// TwinCAT 3 PLC project CORE
// Title: ZigaLibs.Core
// Company: Ziga Javornik
// Author: Ziga Javornik
// ProjectVersion: 0.0.3.7
// Description: A collection of core objects for work with further libraries implementations.
// ProgramVersion: 3.1.4026.26
// libraries:
//   Tc2_EtherCAT, * (Beckhoff Automation GmbH)
//   Tc2_IoFunctions, * (Beckhoff Automation GmbH)
//   Tc2_Standard, * (Beckhoff Automation GmbH)
//   Tc2_System, * (Beckhoff Automation GmbH)
//   Tc2_Utilities, * (Beckhoff Automation GmbH)
//   Tc3_Module, * (Beckhoff Automation GmbH)
//   TcError, * (Roald87)
//   TcUnit, * (www.tcunit.org)
//   Base Interfaces,newest,System
// project tree:
//   SOURCE/Array/ ArrayHelper.TcPOU
//   SOURCE/Array/DUTs/ ST_ArrayProperties.TcDUT, T_ArrayIndexer.TcDUT
//   SOURCE/Beckhoff/Ads/ AdsHelper.TcPOU, FB_HasAmsAddressFromProcessImage.TcPOU, I_HasAmsAddress.TcIO
//   SOURCE/Beckhoff/EtherCAT/CoE/DUTs/ ST_CoeEntry.TcDUT, ST_CoeEntry_DINT.TcDUT, ST_CoeEntry_SINT.TcDUT, ST_CoeEntry_String128.TcDUT, ST_CoeEntry_UDINT.TcDUT, ST_CoeEntry_INT.TcDUT, ST_CoeEntry_REAL.TcDUT, ST_CoeEntry_String255.TcDUT, ST_CoeEntry_String30.TcDUT, ST_CoeEntry_UINT.TcDUT, ST_CoeEntry_USINT.TcDUT, T_CoEIndex.TcDUT, T_CoESubIndex.TcDUT
//   SOURCE/Beckhoff/EtherCAT/CoE/ FB_CoeReadWrite.TcPOU, I_ReadsCoE.TcIO
//   SOURCE/Beckhoff/EtherCAT/Diagnosis/DUTs/Device state/ E_EcDeviceState.TcDUT, E_EcDeviceStateExtras.TcDUT, E_EcLinkState.TcDUT, ST_EcDeviceState.TcDUT, ST_EcSlaveState.TcDUT
//   SOURCE/Beckhoff/EtherCAT/Diagnosis/DUTs/ E_EthercatDiagnosisState.TcDUT, E_EthercatDiagnosisStatus.TcDUT, ST_EthercatSlaveInfo.TcDUT
//   SOURCE/Beckhoff/EtherCAT/Diagnosis/ FB_EthercatDiagnosis.TcPOU (excluded from build), I_EthercatDiagnosis.TcIO
//   SOURCE/Beckhoff/EtherCAT/ EthercatHelper.TcPOU, FB_ReadBoxName.TcPOU
//   SOURCE/Errors/DUTs/ ST_AdsError.TcDUT, ST_Error.TcDUT, ST_GenericError.TcDUT
//   SOURCE/Errors/ FB_ErrorSource.TcPOU, I_HasError.TcIO, I_ErrorSource.TcIO, I_HasAdsError.TcIO, I_HasGenericError.TcIO
//   SOURCE/General/ FB_BooleanObserver.TcPOU, FB_HasInstanceNameAndPath.TcPOU, FB_HasTaskInfo.TcPOU, FB_Watchdog.TcPOU, InstanceNameHelper.TcPOU, ST_Value.TcDUT (not stored)
//   SOURCE/General/Memory/ FB_Malloc.TcPOU, MemoryHelper.TcPOU, ST_AllocatedMemoryProperties.TcDUT, E_MemCmpResults.TcDUT
//   SOURCE/General/Variable information/ T_VarInfo.TcDUT, F_DoesVarTypeEqual.TcPOU, F_GetVarInfo.TcPOU, ST_VarInfo.TcDUT, T_VarSize.TcDUT
//   SOURCE/General/Variable extensions/ BoolEx.TcPOU
//   SOURCE/String/StringBuilder/Extensions/AddAny/ E_AddAnyBitOptions.TcDUT, I_StringBuilderEx_Any.TcIO
//   SOURCE/String/StringBuilder/ FB_StringBuilder.TcPOU, I_StringBuilder.TcIO
//   SOURCE/String/ StringConstants.TcPOU, StringHelper.TcPOU, T_Char.TcDUT
//   SOURCE/Time/DUTs/ E_TimeFormat.TcDUT (not stored), ST_CurrentSystemTimeInfo.TcDUT
//   SOURCE/Time/ FB_DateTimeToStringConverter.TcPOU, FB_LocalSystemTimeProvider.TcPOU, I_DateTimeToStringConverter.TcIO, I_LocalSystemTimeProvider.TcIO
//   / TestsTask.TcTTO
//   TESTS/ PRG_TESTS.TcPOU
//   TESTS/Test suites/ FB_AdsHelper_Tests.TcPOU, FB_ArrayHelper_Tests.TcPOU, FB_CoeReadWrite_Tests.TcPOU, FB_DateTimeToStringConverter_Tests.TcPOU, FB_ErrorSource_ExtensionForTests.TcPOU, FB_ErrorSource_Tests.TcPOU, FB_EthercatDiagnosis_Tests.TcPOU (excluded from build), FB_EthercatHelper_Tests.TcPOU, FB_HasInstanceName_ExtensionForTests.TcPOU, FB_HasInstanceName_Tests.TcPOU, FB_HasTaskInfo_ExtensionsForTests.TcPOU, FB_HasTaskInfo_Tests.TcPOU, FB_Malloc_Tests.TcPOU, FB_StringBuilderEx_Any_Tests.TcPOU, FB_StringBuilder_Tests.TcPOU, FB_BoolEx_Tests.TcPOU, FB_StringHelper_Tests.TcPOU
//   TESTS/Test suites/Time/ FB_LocalSystemTime_Tests.TcPOU
// (motion and I/O tree: see PLC project logging)
// real-time tasks:
//   TASK TestsTask: cycle T#10ms, priority 20, ADS port 350
//   TASK PlcTask: cycle T#10ms, priority 21, ADS port 351

CONFIGURATION CORE
    RESOURCE PLC ON TwinCAT3
        TASK TestsTask(INTERVAL := T#10ms, PRIORITY := 20);
        PROGRAM PRG_TESTS WITH TestsTask : PRG_TESTS;
    END_RESOURCE
END_CONFIGURATION

// ---- SOURCE/Array/DUTs/ST_ArrayProperties.TcDUT
TYPE ST_ArrayProperties :
STRUCT
	Count		: DINT;
	StartIndex	: T_ArrayIndexer;
	EndIndex	: T_ArrayIndexer;
END_STRUCT
END_TYPE

// ---- SOURCE/Array/DUTs/T_ArrayIndexer.TcDUT
// Should be used when accessing array index.
TYPE T_ArrayIndexer : DINT; END_TYPE

// ---- SOURCE/Beckhoff/EtherCAT/CoE/DUTs/ST_CoeEntry.TcDUT
{attribute 'qualified_only'}
// CoE entry in the dictionary, includes index and the subindex
TYPE ST_CoeEntry :
STRUCT
	Index		: T_CoEIndex;
	Subindex	: T_CoESubIndex;
END_STRUCT
END_TYPE

// ---- SOURCE/Beckhoff/EtherCAT/CoE/DUTs/ST_CoeEntry_DINT.TcDUT
TYPE ST_CoeEntry_DINT EXTENDS ST_CoeEntry :
STRUCT
	Value	: DINT;
END_STRUCT
END_TYPE

// ---- SOURCE/Beckhoff/EtherCAT/CoE/DUTs/ST_CoeEntry_SINT.TcDUT
TYPE ST_CoeEntry_SINT EXTENDS ST_CoeEntry :
STRUCT
	Value	: SINT;
END_STRUCT
END_TYPE

// ---- SOURCE/Beckhoff/EtherCAT/CoE/DUTs/ST_CoeEntry_String128.TcDUT
TYPE ST_CoeEntry_String128 EXTENDS ST_CoeEntry :
STRUCT
	Value	: STRING(128);
END_STRUCT
END_TYPE

// ---- SOURCE/Beckhoff/EtherCAT/CoE/DUTs/ST_CoeEntry_UDINT.TcDUT
TYPE ST_CoeEntry_UDINT EXTENDS ST_CoeEntry :
STRUCT
	Value	: UDINT;
END_STRUCT
END_TYPE

// ---- SOURCE/Beckhoff/EtherCAT/CoE/DUTs/ST_CoeEntry_INT.TcDUT
TYPE ST_CoeEntry_INT EXTENDS ST_CoeEntry :
STRUCT
	Value	: INT;
END_STRUCT
END_TYPE

// ---- SOURCE/Beckhoff/EtherCAT/CoE/DUTs/ST_CoeEntry_REAL.TcDUT
TYPE ST_CoeEntry_REAL EXTENDS ST_CoeEntry :
STRUCT
	Value	: REAL;
END_STRUCT
END_TYPE

// ---- SOURCE/Beckhoff/EtherCAT/CoE/DUTs/ST_CoeEntry_String255.TcDUT
TYPE ST_CoeEntry_String255 EXTENDS ST_CoeEntry :
STRUCT
	Value	: Tc2_System.T_MaxString;
END_STRUCT
END_TYPE

// ---- SOURCE/Beckhoff/EtherCAT/CoE/DUTs/ST_CoeEntry_String30.TcDUT
TYPE ST_CoeEntry_String30 EXTENDS ST_CoeEntry :
STRUCT
	Value	: STRING(30);
END_STRUCT
END_TYPE

// ---- SOURCE/Beckhoff/EtherCAT/CoE/DUTs/ST_CoeEntry_UINT.TcDUT
TYPE ST_CoeEntry_UINT EXTENDS ST_CoeEntry :
STRUCT
	Value	: UINT;
END_STRUCT
END_TYPE

// ---- SOURCE/Beckhoff/EtherCAT/CoE/DUTs/ST_CoeEntry_USINT.TcDUT
TYPE ST_CoeEntry_USINT EXTENDS ST_CoeEntry :
STRUCT
	Value	: USINT;
END_STRUCT
END_TYPE

// ---- SOURCE/Beckhoff/EtherCAT/CoE/DUTs/T_CoEIndex.TcDUT
TYPE T_CoEIndex : WORD; END_TYPE

// ---- SOURCE/Beckhoff/EtherCAT/CoE/DUTs/T_CoESubIndex.TcDUT
TYPE T_CoESubIndex : BYTE; END_TYPE

// ---- SOURCE/Beckhoff/EtherCAT/Diagnosis/DUTs/Device state/E_EcDeviceState.TcDUT
{attribute 'qualified_only'}
TYPE E_EcDeviceState :
(
	INIT		:= Tc2_EtherCAT.EC_DEVICE_STATE_INIT,
	PREOP		:= Tc2_EtherCAT.EC_DEVICE_STATE_PREOP,
	BOOTSTRAP	:= Tc2_EtherCAT.EC_DEVICE_STATE_BOOTSTRAP,
	SAFEOP		:= Tc2_EtherCAT.EC_DEVICE_STATE_SAFEOP,
	OP			:= Tc2_EtherCAT.EC_DEVICE_STATE_OP
)BYTE;
END_TYPE

// ---- SOURCE/Beckhoff/EtherCAT/Diagnosis/DUTs/Device state/E_EcDeviceStateExtras.TcDUT
{attribute 'qualified_only'}
TYPE E_EcDeviceStateExtras :
(
	NOTHING				:= 16#00,
	STATE_MACHINE_ERROR := Tc2_EtherCAT.EC_DEVICE_STATE_ERROR,
	INVALID_VPRS		:= Tc2_EtherCAT.EC_DEVICE_STATE_INVALID_VPRS,
	INIIT_CMD_ERROR		:= Tc2_EtherCAT.EC_DEVICE_STATE_INITCMD_ERROR,
	DISABLED			:= Tc2_EtherCAT.EC_DEVICE_STATE_DISABLED
)BYTE;
END_TYPE

// ---- SOURCE/Beckhoff/EtherCAT/Diagnosis/DUTs/Device state/E_EcLinkState.TcDUT
TYPE E_EcLinkState :
(
	OK					:= Tc2_EtherCAT.EC_LINK_STATE_OK,
	NOT_PRESENT			:= Tc2_EtherCAT.EC_LINK_STATE_NOT_PRESENT,
	LINK_WITHOUT_COMM	:= Tc2_EtherCAT.EC_LINK_STATE_LINK_WITHOUT_COMM,
	MISSING_LINK		:= Tc2_EtherCAT.EC_LINK_STATE_MISSING_LINK,
	ADDITIONAL_LINK		:= Tc2_EtherCAT.EC_LINK_STATE_ADDITIONAL_LINK,
	PORT_A				:= Tc2_EtherCAT.EC_LINK_STATE_PORT_A,
	PORT_B				:= Tc2_EtherCAT.EC_LINK_STATE_PORT_B,
	PORT_C				:= Tc2_EtherCAT.EC_LINK_STATE_PORT_C,
	PORT_D				:= Tc2_EtherCAT.EC_LINK_STATE_PORT_D
)BYTE;
END_TYPE

// ---- SOURCE/Beckhoff/EtherCAT/Diagnosis/DUTs/Device state/ST_EcDeviceState.TcDUT
TYPE ST_EcDeviceState :
STRUCT
	State		: E_EcDeviceState;	// Device state
	StateExtras	: E_EcDeviceStateExtras;	// Extra information
END_STRUCT
END_TYPE

// ---- SOURCE/Beckhoff/EtherCAT/Diagnosis/DUTs/Device state/ST_EcSlaveState.TcDUT
TYPE ST_EcSlaveState :
STRUCT
	Device	: ST_EcDeviceState;	// Device state
	Link	: E_EcLinkState;	// Link state
END_STRUCT
END_TYPE

// ---- SOURCE/Beckhoff/EtherCAT/Diagnosis/DUTs/E_EthercatDiagnosisState.TcDUT
{attribute 'qualified_only'}
{attribute 'strict'}
TYPE E_EthercatDiagnosisState :
(
	READY,
	GET_SLAVE_STATES,
	GET_FAULTY_SLAVE_ADDRESSES,
	FINISHED,
	ERROR
);
END_TYPE

// ---- SOURCE/Beckhoff/EtherCAT/Diagnosis/DUTs/E_EthercatDiagnosisStatus.TcDUT
TYPE E_EthercatDiagnosisStatus :
(
	NO_ERROR,				// No error, all slaves are present
	MISSING_ALLOWED_SLAVES,	// Missing slaves, but they are allowed (for example, hot connect)
	ERROR					// Missing slaves that are not allowed to be missing
);
END_TYPE

// ---- SOURCE/Beckhoff/EtherCAT/Diagnosis/DUTs/ST_EthercatSlaveInfo.TcDUT
TYPE ST_EthercatSlaveInfo :
STRUCT
	Name		: Tc2_System.T_MaxString;	// Slave name
	IsIgnored	: BOOL;	// True if slave is ignored with the scan
	State		: ST_EcSlaveState;
END_STRUCT
END_TYPE

// ---- SOURCE/Errors/DUTs/ST_AdsError.TcDUT
TYPE ST_AdsError EXTENDS ST_Error:
STRUCT
	Code	: TcError.AdsErrorCodes;
	Message	: Tc2_System.T_MaxString;
END_STRUCT
END_TYPE

// ---- SOURCE/Errors/DUTs/ST_Error.TcDUT
TYPE ST_Error :
STRUCT
	Source	: Tc2_System.T_MaxString;
END_STRUCT
END_TYPE

// ---- SOURCE/Errors/DUTs/ST_GenericError.TcDUT
TYPE ST_GenericError EXTENDS ST_Error :
STRUCT
	Code	: DINT;
	Message	: Tc2_System.T_MaxString;
END_STRUCT
END_TYPE

// ---- SOURCE/General/Memory/ST_AllocatedMemoryProperties.TcDUT
// Properties for working with dynamic memory allocation.
TYPE ST_AllocatedMemoryProperties :
STRUCT
	Size				: DINT;		// Size of the allocated memory
	StartAddress		: PVOID;	// Pointer to the address of the array memory space
	BaseTypeSize		: DINT;		// Size of the base type provided, when allocated
	NumberOfElements	: DINT;	// Number of elements provided, when allocated.
END_STRUCT
END_TYPE

// ---- SOURCE/General/Variable information/T_VarInfo.TcDUT
TYPE T_VarInfo : __SYSTEM.VAR_INFO; END_TYPE

// ---- SOURCE/General/Memory/E_MemCmpResults.TcDUT
{attribute 'qualified_only'}
TYPE E_MemCmpResults :
(
	pBUFF1_LESS_THAN_pBUFF2	:= -1,
	IDENTICAL	:= 0,
	PbUFF1_GREATER_THAN_pBUFF2	:= 1,
	ERROR	:= 255
)DINT;
END_TYPE

// ---- SOURCE/General/Variable information/ST_VarInfo.TcDUT
TYPE ST_VarInfo :
STRUCT
	DataType	: __SYSTEM.TYPE_CLASS;
	Address		: POINTER TO BYTE;
	Size		: T_VarSize;
END_STRUCT
END_TYPE

// ---- SOURCE/General/Variable information/T_VarSize.TcDUT
// Variable size alias type. To be used when working with SIZEOF operator.
TYPE T_VarSize : UXINT; END_TYPE

// ---- SOURCE/String/StringBuilder/Extensions/AddAny/E_AddAnyBitOptions.TcDUT
{attribute 'qualified_only'}
{attribute 'strict'}
// Provides various options of how ANY_BIT data type can be converted.
TYPE E_AddAnyBitOptions :
(
	BINARY,			// Will be converted to a binary string (base 2)
	DECIMAL,		// Will be converted to a decial string (base 10)
	HEXADECIMAL,	// Will be converted to hexadecimal string (base 16)
	OCTAL			// Will be converted to octal string (base 8)
);
END_TYPE

// ---- SOURCE/String/T_Char.TcDUT
TYPE T_Char : STrING(1); END_TYPE

// ---- SOURCE/Time/DUTs/ST_CurrentSystemTimeInfo.TcDUT
TYPE ST_CurrentSystemTimeInfo :
STRUCT
	IsValid	: BOOL;
	Value	: Tc2_Utilities.TIMESTRUCT;
END_STRUCT
END_TYPE

// ---- SOURCE/Beckhoff/Ads/I_HasAmsAddress.TcIO
// Interface to implement when requiring AMS address
INTERFACE I_HasAmsAddress

// Gets or sets the Ams address structure
PROPERTY AmsAddress : REFERENCE TO Tc2_System.ST_AmsAddr
GET
END_GET
SET
END_SET
END_PROPERTY

END_INTERFACE

// ---- SOURCE/Beckhoff/EtherCAT/CoE/I_ReadsCoE.TcIO
INTERFACE I_ReadsCoE

// Reads CoE items and updates them. Returns TRUE when done,
// Needs to be called until the method finishes, indicating via the return value. 
METHOD PUBLIC ReadCoE : BOOL
END_METHOD

END_INTERFACE

// ---- SOURCE/Beckhoff/EtherCAT/Diagnosis/I_EthercatDiagnosis.TcIO
INTERFACE I_EthercatDiagnosis

// Returns TRUE if an error occurred while performing the scan
PROPERTY Error : BOOL
GET
END_GET
END_PROPERTY

// Gets an array of slaves that have been added to ignore list
PROPERTY IgnoredSlaves : REFERENCE TO ARRAY[0..255] OF Tc2_System.T_MaxString
GET
END_GET
END_PROPERTY

// Adds the provided slave to a collection of slaves that will not trigger an error
// Example is slaves that are used on hot connect groups, and when connected should not cause an error. 
METHOD IgnoreSlave
VAR_INPUT
	Name	: Tc2_System.T_MaxString;	// Slave to be ignored if not found or an error is reported back
END_VAR
END_METHOD

// Returns an array of misisng slave names
PROPERTY MissingSlaves : REFERENCE TO ARRAY[0..255] OF ST_EthercatSlaveInfo
GET
END_GET
END_PROPERTY

// Reset the internal state machine of diagnosis and clearing any errors, if active.
METHOD Reset
END_METHOD

// Performs a scan on the EtherCAT master, returns TRUE when done.
METHOD Scan	: BOOL
VAR_INPUT
	EcMasterNetId	: AMSNETID;
END_VAR
END_METHOD

// Gets the status based on last executed scan.
PROPERTY Status : E_EthercatDiagnosisStatus
GET
END_GET
END_PROPERTY

END_INTERFACE

// ---- SOURCE/Errors/I_HasError.TcIO
INTERFACE I_HasError

{attribute 'monitoring':='call'}
// Returns TRUE if an error has occurred
PROPERTY Error : BOOL
GET
END_GET
END_PROPERTY

END_INTERFACE

// ---- SOURCE/Errors/I_ErrorSource.TcIO
INTERFACE I_ErrorSource EXTENDS I_HasAdsError, I_HasGenericError, I_HasError

END_INTERFACE

// ---- SOURCE/Errors/I_HasAdsError.TcIO
INTERFACE I_HasAdsError

{attribute 'monitoring':='call'}
// Gets or sets the Ads error - note that code to message conversion is done automatically.
PROPERTY AdsError : REFERENCE TO ST_AdsError
GET
END_GET
END_PROPERTY

END_INTERFACE

// ---- SOURCE/Errors/I_HasGenericError.TcIO
INTERFACE I_HasGenericError

{attribute 'monitoring':='call'}
// Gets the Generic error
PROPERTY GenericError : REFERENCE TO ST_GenericError
GET
END_GET
END_PROPERTY

END_INTERFACE

// ---- SOURCE/String/StringBuilder/Extensions/AddAny/I_StringBuilderEx_Any.TcIO
INTERFACE I_StringBuilderEx_Any

(* Adds the variable of any data type to the sequence. Conversion is done automatically from within.
Some extra info: 
	- BOOL and BIT will have the string converted to 'TRUE' and 'FALSE' respectively.
	- floating point variables will have their values precision based on constructor realFormatPrecision and will be rounded based on the roundRealValues
*)
METHOD AddAny : REFERENCE TO FB_StringBuilder
VAR_INPUT
	anyVar	: ANY;
END_VAR
END_METHOD

// Adds a variable of type ANY_BIT to the string generating sequence, based on the provided parameters.
// This includes: BYTE, WORD, DWORD, LWORD, 
METHOD AddAnyBit : REFERENCE TO FB_StringBuilder
VAR_INPUT
	anyBit					: ANY_BIT;				// Value to be converterd
	option					: E_AddAnyBitOptions;	// Select how the value is converter
	lowerCase				: BOOL;					// If hexadecimal option is selected, the result string can be converted to either lower or upper case
	displayedDigitsCount	: INT;					// This determines how many digits are to be displayed. If actual digits count is lower, the string is filled with zeros from the left side. If left at 0, the result string will be an empty string!
	addNotation				: BOOL;					// If this is set to TRUE, a notation will be prepended: (DEC)10, (BIN)10, (HEX)10, (OCT)10
END_VAR
END_METHOD

// Adds any REAL or LREAL value to the generating string sequence.
// Please note that REAL values will ALWAYS be automatically rounded on 3rd decimal digit.
// Anything after it will be whatever TwinCAT representation decides to do.
METHOD AddAnyReal : REFERENCE TO FB_StringBuilder
VAR_INPUT
	anyReal		: ANY_REAL;	// Value to be converter
	precision	: INT;		// Precision
	round		: BOOL;		// Rounding of the last displayed digit
END_VAR
END_METHOD

END_INTERFACE

// ---- SOURCE/String/StringBuilder/I_StringBuilder.TcIO
INTERFACE I_StringBuilder

// Adds a string to the build sequence.
METHOD AddString : REFERENCE TO FB_StringBuilder
VAR_INPUT
	str	: Tc2_System.T_MaxString;	// String to be added.
END_VAR
END_METHOD

// Adds a string to the build sequence and wraps the str in double quotation marks "str"
METHOD AddWithDblQuotationMarks : REFERENCE TO FB_StringBuilder
VAR_INPUT
	str : Tc2_System.T_MaxString;
END_VAR
END_METHOD

// Adds a string to the build sequence and wraps the str in quotation marks 'str'
METHOD AddWithQuotationMark : REFERENCE TO FB_StringBuilder
VAR_INPUT
	str	: Tc2_System.T_MaxString;
END_VAR
END_METHOD

// Finishes string generation and returns the generated string
METHOD Create : Tc2_System.T_MaxString
END_METHOD

(* Reset the string build sequence, clear any string built so far.*)
METHOD Reset : REFERENCE TO FB_StringBuilder
VAR_INPUT
END_VAR
END_METHOD

END_INTERFACE

// ---- SOURCE/Time/I_DateTimeToStringConverter.TcIO
INTERFACE I_DateTimeToStringConverter

(* Converts TIMESTRUCT to STRING.*)
METHOD DateTime : STRING
VAR_INPUT
	timeFormat			: E_TimeFormat;	// Time format to apply to the timestruct conversion
	timeOfDaySeperator	: STRING(1);	// Specifies how time of day is split
	dateSeperator		: STRING(1);	// Specifies how date is split
	fillWithZeros		: BOOL;	// If set to true: month, day hour, minute and second will have 0 added when only a single digit is present
	IncludeMilliseconds	: BOOL; // If set to true, milliseconds will also be displayed in the result, else they are ignored
END_VAR
END_METHOD

(* Converts TIMESTRUCT.wDay to STRING.*)
METHOD Day : STRING
VAR_INPUT
	fillWithZeros	: BOOL;	// If set to true, result will have 0 added when only a single digit is present
END_VAR
END_METHOD

(* Converts TIMESTRUCT.wHour to STRING.*)
METHOD Hour : STRING
VAR_INPUT
	fillWithZeros	: BOOL;	// If set to true, result will have 0 added when only a single digit is present
END_VAR
END_METHOD

(* Converts TIMESTRUCT.wMillisecond to STRING.*)
METHOD Millisecond : STRING
VAR_INPUT
	fillWithZeros	: BOOL;	// If set to true, result will have 0 added when only a single digit is present
END_VAR
END_METHOD

(* Converts TIMESTRUCT.wMinute to STRING.*)
METHOD Minute : STRING
VAR_INPUT
	fillWithZeros	: BOOL;	// If set to true, result will have 0 added when only a single digit is present
END_VAR
END_METHOD

(* Converts TIMESTRUCT.wMonth to STRING.*)
METHOD Month : STRING
VAR_INPUT
	fillWithZeros	: BOOL;	// If set to true, result will have 0 added when only a single digit is present
END_VAR
END_METHOD

(* Converts TIMESTRUCT.wSecond to STRING.*)
METHOD Second : STRING
VAR_INPUT
	fillWithZeros	: BOOL;	// If set to true, result will have 0 added when only a single digit is present
END_VAR
END_METHOD

(* Converts TIMESTRUCT.wYear to STRING.*)
METHOD Year : STRING
END_METHOD

END_INTERFACE

// ---- SOURCE/Time/I_LocalSystemTimeProvider.TcIO
INTERFACE I_LocalSystemTimeProvider

METHOD PUBLIC ConvertToString : I_DateTimeToStringConverter
VAR_INPUT
END_VAR
END_METHOD

{attribute 'monitoring':='call'}
// Gets current system timo info as a <ST_CurrentSystemTimeInfo>
PROPERTY CurrentTime : REFERENCE TO ST_CurrentSystemTimeInfo
GET
END_GET
END_PROPERTY

END_INTERFACE

// ---- TESTS/PRG_TESTS.TcPOU
PROGRAM INTERNAL PRG_TESTS

(* Instantiate test suites here. Naming convention for tests should be a suffix with _Tests.
Good practice for creating test methods is to end them with _test as well. *)
VAR
	AdsHelperTests					: FB_AdsHelper_Tests;
	ArrayHelperTests				: FB_ArrayHelper_Tests;
	DateTimeToStringConverterTest	: FB_DateTimeToStringConverter_Tests;
	ErrorSourceTests				: FB_ErrorSource_Tests;
	HasInstanceNameTests			: FB_HasInstanceName_Tests;
	StringBuilderTests				: FB_StringBuilder_Tests;
	HasTaskInfoTests				: FB_HasTaskInfo_Tests;
	BoolExTests						: FB_BoolEx_Tests;
	EthercatHelperTests				: FB_EthercatHelper_Tests;
	//EthercatDiagnosisTests			: FB_EthercatDiagnosis_Tests;
	MallocTests						: FB_Malloc_Tests;
	StringHelperTests				: FB_StringHelper_Tests;
	LocalSystemTimeTests			: FB_LocalSystemTime_Tests;
	CoeReadWriteTests				: FB_CoeReadWrite_Tests;
END_VAR

// Run tests in paralel
//TcUnit.RUN();

// Run tests in sequence, one after the other. Uncomment if required.
TcUnit.RUN_IN_SEQUENCE();

END_PROGRAM

// ---- TESTS/Test suites/FB_AdsHelper_Tests.TcPOU
// Subject under test
FUNCTION_BLOCK INTERNAL FB_AdsHelper_Tests EXTENDS FB_TestSuite

// Create instance variables that will be accesible for all tests
VAR
END_VAR

// Call your test methods here
Test_NetIdToString_AllZeros_ExpectEmptyString();
Test_MasterAddress();

METHOD Test_MasterAddress

VAR_INST
	masterNetId	: Tc2_System.T_AmsNetID := '0.0.0.0.0.5';
END_VAR
TcUnit.TEST('Test_MasterAddress');

AssertEquals_DINT(
	Expected := 24,
	Actual := 24,
	Message := 'Getting address from master netId was incorrect!');
	
TcUnit.TEST_FINISHED();
END_METHOD

METHOD PRIVATE Test_NetIdToString_AllZeros_ExpectEmptyString

(* Instanced variables are VERY useful for writing tests since tests are run in paralel (by default).
By instantiating local variables that are not placed on the same stack as method (values are retained between calls)
you make sure that the SUT is not changed by some other test. *)
VAR_INST
	
END_VAR

// Place temporary variables here
VAR
	emptyNetId	: Tc2_System.T_AmsNetIdArr;
END_VAR
// The name of the test, is the same as method name!
TcUnit.TEST('Test_NetIdToString_AllZeros_ExpectEmptyString');

// Do your assertions here...
AssertEquals_STRING(
	Expected := '',
	Actual := AdsHelper.NetIdToString(emptyNetId),
	Message := 'An empty netId should return an empty string!');

TcUnit.TEST_FINISHED();
END_METHOD

END_FUNCTION_BLOCK

// ---- SOURCE/Beckhoff/Ads/AdsHelper.TcPOU
// A helper class providing various helpful methods when working with ads data
PROGRAM AdsHelper

// Returns last part of the netId, which is the ID of the etherCAT master.
METHOD PUBLIC GetEthercatMasterIdFromNetIdString : UDINT
VAR_INPUT
	netId	: Tc2_System.T_AmsNetID;
END_VAR

VAR
	sNetIdResult	: T_AmsNetID;
	nMasterAddress	: UDINT;
	nDotPosition	: INT;
END_VAR
sNetIdResult := netId;
nDotPosition := Tc2_Standard.FIND(sNetIdResult, '.');

WHILE nDotPosition <> 0 DO
	nDotPosition := Tc2_Standard.FIND(sNetIdResult, '.');
	IF nDotPosition = 0 THEN
		EXIT;
	END_IF
	sNetIdResult := Tc2_Standard.DELETE(STR := sNetIdResult, POS := 1, LEN := nDotPosition);
END_WHILE

GetEthercatMasterIdFromNetIdString := STRING_TO_UDINT(sNetIdResult);
END_METHOD

// Converts netId of type <Tc2_System.T_AmsNetIdArr> to <T_AmsNetID>, which equates to <STRING(23)>.
METHOD PUBLIC NetIdToString : T_AmsNetID
VAR_INPUT
	netId	: Tc2_System.T_AmsNetIdArr;	// NetId to be converted
END_VAR

VAR
	arrayMaxIndex	: DINT;
	i				: DINT;
END_VAR
arrayMaxIndex := ArrayHelper.GetMaxIndex(
	arr := netId, 
	dataType := netId[0], 
	startIndex := 0);

FOR i := 0 TO arrayMaxIndex BY 1 DO
	// If any element is not 0, exit and call the system function to convert
	IF netId[i] <> 0 THEN
		EXIT;
	END_IF
	// If reaching last element in the array, this means only 0s are present, indicating local netId - return empty string
	IF i = ArrayHelper.GetMaxIndex(arr := netId, dataType := netId[0], startIndex := 0) THEN
		NetIdToString := '';
		RETURN;
	END_IF
END_FOR

NetIdToString := Tc2_System.F_CreateAmsNetId(nIds := netId);
END_METHOD

END_PROGRAM

// ---- SOURCE/Array/ArrayHelper.TcPOU
{attribute 'enable_dynamic_creation'}
// Provides array helper methods for easier work with arrays accross programming.
PROGRAM ArrayHelper

// Clears the entire array. Returns TRUE if operation was sucessfull.
METHOD PUBLIC Clear : BOOL
VAR_INPUT
	arr			: ANY;	// Array to be cleared
END_VAR
IF NOT ValidateArrayVar(arr) THEN
	RETURN;
END_IF

Tc2_System.MEMSET(
	destAddr := arr.pValue,
	fillByte := 0,
	n := DINT_TO_UDINT(arr.diSize));
	
Clear := TRUE;
END_METHOD

// Looks trough the array and returns TRUE if any element equals to the one provided.
METHOD DoesArrayContainItem : BOOL
VAR_INPUT
	arr		: ANY;	// Array to be checked
	item	: ANY;	// Item to be found in the array
END_VAR

VAR
	itemCount	: T_ArrayIndexer;
	currentItem	: T_ArrayIndexer;
	cmpResult	: E_MemCmpResults;
END_VAR
IF NOT ValidateArrayVar(arr) THEN
	RETURN;
END_IF

IF item.diSize = 0 OR_ELSE	// If item size is 0
	(arr.diSize MOD item.diSize) <> 0 	// If incorrect item is provided (division will return non 0 remainder)
THEN
	RETURN;
END_IF

itemCount := arr.diSize/item.diSize;

FOR currentItem := 0 TO itemCount - 1 BY 1 DO
	cmpResult := Tc2_System.MEMCMP(
		pBuf1 := arr.pValue + DINT_TO_DWORD(currentItem * item.diSize),
		pBuf2 := item.pValue,
		n := DINT_TO_UDINT(item.diSize));
		
	IF cmpResult = E_MemCmpResults.IDENTICAL THEN
		DoesArrayContainItem := TRUE;
		RETURN;
	END_IF
END_FOR
END_METHOD

// Looks trough the array and return the last non-zero element to the result variable.
// Returns TRUE if an element was found and FALSE if no empty elements are found.
// Note that this method uses memmory allocation. All occupied memory is released after method finishes.
METHOD PUBLIC FindLastOccupiedItem	: BOOL
VAR_INPUT
	arr			: ANY;	// Array to look for the last element value
	dataType	: ANY;	// Data type of the array elements, can be used like this : datayType := arr[0]
	result		: ANY;	// Result variable, result be written to this variable
END_VAR

VAR
	i								: T_ArrayIndexer;
	maxIndex						: T_ArrayIndexer;
	compareResult					: E_MemCmpResults;
	ptrAllocatedBytes_emptyElement	: POINTER TO BYTE;
END_VAR
IF NOT ValidateArrayVar(arr) OR result.TypeClass <> dataType.TypeClass THEN
	RETURN;
END_IF

maxIndex :=  GetElementCount(arr := arr, dataType := dataType) - 1;
ptrAllocatedBytes_emptyElement := __NEW(BYTE, DINT_TO_UDINT(dataType.diSize));

// Array with 1 element - loop would point to invalid position, exit early by just checking the values
IF maxIndex = 0 THEN
	IF arr.pValue^ <> ptrAllocatedBytes_emptyElement^ THEN
		Tc2_System.MEMCPY(
			srcAddr := arr.pValue,
			destAddr := result.pValue,
			n := DINT_TO_UDINT(dataType.diSize));
			FindLastOccupiedItem := TRUE;
	END_IF
	// Delete allocated memory and return from the method
	__DELETE(ptrAllocatedBytes_emptyElement);
	RETURN;
END_IF

FOR i := maxIndex TO 0 BY -1 DO
	compareResult := Tc2_System.MEMCMP(
		pBuf1 := arr.pValue +  DINT_TO_DWORD(i * dataType.diSize),
		pBuf2 := ptrAllocatedBytes_emptyElement,
		n := DINT_TO_UDINT(dataType.diSize));
		
	// If element is not empty, return
	IF compareResult <> E_MemCmpResults.IDENTICAL THEN
		Tc2_System.MEMCPY(
			srcAddr := arr.pValue +  DINT_TO_DWORD(i * dataType.diSize),
			destAddr := result.pValue,
			n := DINT_TO_UDINT(dataType.diSize));
		FindLastOccupiedItem := TRUE;
		EXIT;
	END_IF
END_FOR

// Delete allocated memory
__DELETE(ptrAllocatedBytes_emptyElement);
END_METHOD

// Returns the number of elements in the array.
METHOD PUBLIC GetElementCount : DINT
VAR_INPUT
	arr			: ANY;	// Array to be checked.
	dataType	: ANY;	// Data type of the array elements, can be used like this : datayType := arr[0]
END_VAR
IF ValidateArrayVar(arr) = FALSE THEN
	RETURN;
END_IF

IF dataType.diSize = 0 THEN
	RETURN;
END_IF
GetElementCount := arr.diSize / dataType.diSize;
END_METHOD

// Gets the maximum array index that can be used for looping or index accessing
METHOD PUBLIC GetMaxIndex : DINT
VAR_INPUT
	arr			: ANY;	// Array to be checked.
	dataType	: ANY;	// Data type of the array elements, can be used like this : datayType := arr[0]
	startIndex	: T_ArrayIndexer;
END_VAR
IF ValidateArrayVar(arr) = FALSE THEN
	RETURN;
END_IF

GetMaxIndex := startIndex + GetElementCount(arr := arr, dataType := dataType) - 1;
END_METHOD

// Inserts the item to the start of the array. 
// Array contents are shifted by 1, last item is deleted.
METHOD InsertAtStart : BOOL
VAR_INPUT	
	arr		: ANY;	// Array to be checked.
	item	: ANY;	// Item to be inserted on start
 END_VAR
IF ValidateArrayVar(arr) = FALSE THEN
	RETURN;
END_IF

ShiftUp(
	arr := arr,
	dataType := item);

// Set first element value
Tc2_System.MEMCPY(
	destAddr := arr.pValue,
	srcAddr := item.pValue,
	n := DINT_TO_UDINT(item.diSize));
END_METHOD

// Iterates the array and sets the value when first empty slot is found. 
// Note that this method uses memmory allocation. All occupied memory is released after method finishes.
METHOD SetAtFirstEmptySlot
VAR_INPUT
	arr		: ANY;	// Array to be checked.
	item	: ANY;	// Item to set
END_VAR

VAR
	ptrByte 			: POINTER TO BYTE;
	i					: T_ArrayIndexer;
	maxIndex			: T_ArrayIndexer;
	ptrAllocatedBytes	: POINTER TO BYTE;
	cmpResult			: DINT;
END_VAR
IF ValidateArrayVar(arr) = FALSE THEN
	RETURN;
END_IF

maxIndex :=  GetElementCount(arr := arr, dataType := item) - 1;
ptrAllocatedBytes := __NEW(BYTE, DINT_TO_UDINT(arr.diSize));

FOR i := 0 TO maxIndex BY 1 DO
	ptrByte := arr.pValue + DINT_TO_UDINT(item.diSize * i);	
	
	cmpResult := Tc2_System.MEMCMP(
			n := DINT_TO_UDINT(item.diSize),
			pBuf1 := ptrAllocatedBytes,
			pBuf2 := ptrByte);
			
	IF cmpResult = E_MemCmpResults.IDENTICAL THEN
		Tc2_System.MEMCPY(
			destAddr := ptrByte,
			n := DINT_TO_UDINT(item.diSize),
			srcAddr := item.pValue);
		EXIT;
	END_IF
END_FOR

__DELETE(ptrAllocatedBytes);
END_METHOD

// Shifts the array down, losing first element and clearing last element in the process.
METHOD ShiftDown
VAR_INPUT
	arr		: ANY;	// Array to be checked.
	dataType	: ANY;	// Data type of the array elements, can be used like this : datayType := arr[0]
END_VAR
IF ValidateArrayVar(arr) = FALSE THEN
	RETURN;
END_IF

Tc2_System.MEMMOVE(	
	destAddr := arr.pValue,
	srcAddr := arr.pValue + DINT_TO_UDINT(dataType.diSize),
	n := DINT_TO_UDINT(arr.diSize - dataType.diSize));

// Clear last element
Tc2_System.MEMSET(
	fillByte := 0,
	n := DINT_TO_UDINT(dataType.diSize),
	destAddr := arr.pValue + DINT_TO_UDINT(arr.diSize - dataType.diSize));
END_METHOD

// Shifts the array up, losing last element and clearing first element in the process.
METHOD ShiftUp
VAR_INPUT
	arr			: ANY;	// Array to be checked.
	dataType	: ANY;	// Data type of the array elements, can be used like this : datayType := arr[0]
END_VAR
IF ValidateArrayVar(arr) = FALSE THEN
	RETURN;
END_IF


Tc2_System.MEMMOVE(
	destAddr := arr.pValue + DINT_TO_UDINT(dataType.diSize),
	srcAddr := arr.pValue,
	n := DINT_TO_UDINT(arr.diSize - dataType.diSize));

// Clear first element
Tc2_System.MEMSET(
	fillByte := 0,
	n := DINT_TO_UDINT(dataType.diSize),
	destAddr := arr.pValue);
END_METHOD

METHOD PRIVATE ValidateArrayVar : BOOL
VAR_INPUT
	arr	: ANY;
END_VAR
VAR
	isArray		: BOOL;
	isReference	: BOOL;
END_VAR
isArray := F_DoesVarTypeEqual(arr, IBaseLibrary.TYPE_ARRAY);
isReference := F_DoesVarTypeEqual(arr, IBaseLibrary.TYPE_REFERENCE);

ValidateArrayVar := isArray OR isReference;
END_METHOD

END_PROGRAM

// ---- SOURCE/General/Variable information/F_DoesVarTypeEqual.TcPOU
// Returns TRUE if the variable's data type equals to the .
FUNCTION F_DoesVarTypeEqual : BOOL
VAR_INPUT
	variable	: ANY;
	typeClass	: IBaseLibrary.TypeClass;
END_VAR
VAR
END_VAR

F_DoesVarTypeEqual := UDINT_TO_INT(variable.TypeClass) = typeClass;

END_FUNCTION

// ---- TESTS/Test suites/FB_ArrayHelper_Tests.TcPOU
FUNCTION_BLOCK INTERNAL FB_ArrayHelper_Tests EXTENDS FB_TestSuite
VAR_INPUT
END_VAR
VAR_OUTPUT
END_VAR

Test01_GetArrayElementCount();
Test02_GetArrayMaxIndex();
Test03_InsertNumber();
Test04_InsertString();
Test05_InsertStruct();
Test06_ShiftUp_ExpectLastElementOverwriteFirstElementZero();
Test07_SetAtFirstEmptySlot();
Test08_AllMethods_provideNonArrayVar_ExpectNothing();
Test09_InsertIntoEmptyArray_ExpectOnlyFirstItem();
Test10_CheckIfArrayContainsItem();
Test11_ClearArray_ExpectEmptyArray();
Test12_ReferenceToArrayWithAllMethods_ExpectNormalResults();
Test13_FindLastOccupiedItem();
Test14_ShiftDown_ExpectFirstElementOverwriteLastElementZero();

METHOD Test01_GetArrayElementCount
VAR_INPUT
END_VAR
VAR
	arr		: ARRAY[0..99] OF REAL;
	arr2	: ARRAY[22..33] OF REAL;
END_VAR
TcUnit.TEST('Test01_GetArrayElementCount');

AssertEquals_DINT(
	Actual := ArrayHelper.GetElementCount(arr := arr, dataType := arr[0]),
	Expected := 100,
	Message := 'Getting array element count failed!');
	
AssertEquals_DINT(
	Actual := ArrayHelper.GetElementCount(arr := arr2, dataType := arr2[22]),
	Expected := 33 - 22 + 1,
	Message := 'Getting array element count for array with non-zero start element index failed!');
	
TcUnit.TEST_FINISHED();
END_METHOD

METHOD Test02_GetArrayMaxIndex
VAR_INPUT
END_VAR
VAR
	arr		: ARRAY[0..99] OF REAL;
	arr2	: ARRAY[22..33] OF REAL;
END_VAR
TcUnit.TEST('Test02_GetArrayMaxIndex');

AssertEquals_DINT(
	Actual := ArrayHelper.GetMaxIndex(arr := arr, dataType := arr[0], startIndex := 0),
	Expected := 99,
	Message := 'Getting array maximum index failed!');
	
AssertEquals_DINT(
	Actual := ArrayHelper.GetMaxIndex(arr := arr2, dataType := arr2[22], startIndex := 22),
	Expected := 33,
	Message := 'Getting array maximum index for array with non-zero start element index failed!');
	
TcUnit.TEST_FINISHED();
END_METHOD

METHOD PRIVATE Test03_InsertNumber
VAR_INPUT
END_VAR

VAR
	i		: INT;
	value	: INT := 99;
	arr		: ARRAY [0..10] OF INT;
END_VAR
TcUnit.TEST('Test03_InsertNumber');

FOR i := 0 TO 10 BY 1 DO
	arr[i] := i;
END_FOR

ArrayHelper.InsertAtStart(
	arr := arr,
	item := value);
	
AssertEquals_INT(
	Expected := value,
	Actual := arr[0],
	Message := 'First item was not inserted properly!');
	
AssertEquals_INT(
	Expected := 9,
	Actual := arr[10],
	Message := 'Last item was not removed from the array!!');
	
TcUnit.TEST_FINISHED();
END_METHOD

METHOD PRIVATE Test04_InsertString
VAR_INPUT
END_VAR

VAR
	i		: INT;
	value	: STRING := '9';
	arr		: ARRAY [0..10] OF STRING;
END_VAR
TcUnit.TEST('Test04_InsertString');

FOR i := 0 TO 10 BY 1 DO
	arr[i] := INT_TO_STRING(i);
END_FOR

ArrayHelper.InsertAtStart(
	arr := arr,
	item := value);
	
AssertEquals_STRING(
 	Actual:= arr[0],
	Expected := value,
	Message := 'First item was not inserted properly!');
	
AssertEquals_STRING(
	Expected := '9',
	Actual := arr[10],
	Message := 'Last item was not removed from the array!!');
	
TcUnit.TEST_FINISHED();
END_METHOD

METHOD Test05_InsertStruct

VAR
	i		: INT;
	value	: ST_GenericError;
	arr		: ARRAY [0..10] OF ST_GenericError;
END_VAR
TcUnit.TEST('Test05_InsertStruct');

FOR i := 0 TO 10 BY 1 DO
	arr[i].Code := i;
	arr[i].Message := INT_TO_STRING(i);
END_FOR

ArrayHelper.InsertAtStart(
	arr := arr,
	item := value);
	
AssertEquals(
	Expected := value,
	Actual := arr[0],
	Message := 'First item was not inserted properly!');
	
AssertEquals_STRING(
	Expected := '9',
	Actual := arr[10].Message,
	Message := 'Last item was not removed from the array!');
	
AssertEquals_STRING(
	Expected := '9',
	Actual := arr[10].Message,
	Message := 'Last item was not removed from the array!');
	
TcUnit.TEST_FINISHED();
END_METHOD

METHOD Test06_ShiftUp_ExpectLastElementOverwriteFirstElementZero
VAR_INPUT
END_VAR

VAR_INST
	arr	: ARRAY[0..20] OF INT;
	i	: int;
END_VAR
TcUnit.TEST('Test06_ShiftUp_ExpectLastElementOverwriteFirstElementZero');

FOR i := 0 TO 20 BY 1 DO
	arr[i] := i;
END_FOR

ArrayHelper.ShiftUp(
	arr := arr,
	dataType := arr[0]);
AssertEquals_INT(
	Actual := arr[0],
	Expected := 0,
	Message := 'Shifting the array up, first element should be set to 0!');
	
FOR i := 1 TO 20 BY 1 DO
	AssertEquals_INT(
		Actual := arr[i],
		Expected := i-1,
		Message := Tc2_Standard.CONCAT('Shifting up failed! Incorrect value at position ', TO_STRING(i)));
END_FOR
	
TcUnit.TEST_FINISHED();
END_METHOD

METHOD Test07_SetAtFirstEmptySlot
VAR_INPUT
END_VAR

VAR
	arr		: ARRAY[0..69] OF T_ArrayIndexer;
	arr2	: ARRAY[0..69] OF BOOL;
	valueToSet	: T_ArrayIndexer := 9999;
	i	: T_ArrayIndexer;
	boolValueToSet	: BOOL := TRUE;
END_VAR
TcUnit.TEST('Test07_SetAtFirstEmptySlot');

FOR i := 0 TO 30 BY 1 DO
	arr[i] := i + 1;
	arr2[i] := TRUE;
END_FOR

ArrayHelper.SetAtFirstEmptySlot(
	arr := arr,
	item := valueToSet);

ArrayHelper.SetAtFirstEmptySlot(
	arr := arr2,
	item := boolValueToSet);

FOR i := 0 TO 30 BY 1 DO
	AssertEquals_DINT(
		Expected := i + 1,
		Actual := arr[i],
		Message := 'Setting first empty slot should not have changed non-empty fields!');
		
	AssertTrue(
		Condition := arr2[i],
		Message := 'Setting first empty slot for array of booleans should not have changed non-empty fields!');
END_FOR

AssertEquals(
	Expected := valueToSet,
	Actual := arr[31],
	Message := 'Setting first empty slot failed, first empty element differs!');
	
AssertTrue(
	Condition := arr2[31],
	Message := 'Setting first empty slot failed, first empty element should be set to TRUE!');
	
AssertEquals_DINT(
	Expected := 0,
	Actual := arr[32],
	Message := 'Setting first empty slot failed, item after the inserted slot should be empty!');
	
AssertFalse(
	Condition := arr2[32],
	Message := 'Setting first empty slot failed, item after the inserted slot should be empty!');	
	

TcUnit.TEST_FINISHED();
END_METHOD

METHOD Test08_AllMethods_provideNonArrayVar_ExpectNothing
VAR_INPUT
END_VAR
VAR
	notAnArray	: BOOL := TRUE;
	val			: BOOL;
END_VAR
TcUnit.TEST('Tes08_AllMethods_provideNonArrayVar_ExpectNothing');

ArrayHelper.GetElementCount(arr := notAnArray, dataType := val);
AssertTrue(
	Condition := notAnArray, 
	Message := 'When non-array is provided to any method, the method should not execute anything!');

AssertEquals_DINT(
	Actual := ArrayHelper.GetMaxIndex(arr := notAnArray, dataType := val, startIndex := 0),
	Expected := 0,
	Message := 'When non-array is provided, max index returned should be 0!');
	
AssertTrue(
	Condition := notAnArray, 
	Message := 'When non-array is provided to any method, the method should not execute anything!');

	
TcUnit.TEST_FINISHED();
END_METHOD

METHOD Test09_InsertIntoEmptyArray_ExpectOnlyFirstItem
VAR_INPUT
END_VAR

VAR_INST
	arr			: ARRAY[0..20] OF ST_GenericError;
	item		: ST_GenericError := (Code := 0, Message := '0');
	emptyItem	: ST_GenericError;
	i 			: T_ArrayIndexer;
END_VAR
TcUnit.TEST('Test09_InsertIntoEmptyArray_ExpectOnlyFirstItem');

FOR i := 0 TO 20 BY 1 DO
	AssertEquals(Actual := arr[i], Expected := emptyItem, Message := 'Wrong array initialization!');
END_FOR

ArrayHelper.InsertAtStart(arr := arr, item := item);

AssertEquals(
	Actual := arr[0], 
	Expected := item, 
	Message := 'InsertAtStart should have first item in array the same as item being inserted!');
	
FOR i := 1 TO 20 BY 1 DO
	AssertEquals(Actual := arr[i], Expected := emptyItem, 
		Message := Tc2_Standard.CONCAT(
			STR1 := 'InsertAtStart should have left other elements unchanged! Changed element at index ', 
			STR2 := TO_STRING(i) ));
END_FOR

ArrayHelper.InsertAtStart(arr := arr, item := item);
AssertEquals(
	Actual := arr[0], 
	Expected := item, 
	Message := 'Inserting at start for the second time - 1st item is incorrect!');
AssertEquals(
	Actual := arr[1], 
	Expected := item, 
	Message := 'Inserting at start for the second time - 2nd item is incorrect!');	

TcUnit.TEST_FINISHED();
END_METHOD

METHOD Test10_CheckIfArrayContainsItem
VAR_INST
	arr		: ARRAY[0..10] OF STRING;
	item	: STRING := 'mwah';
END_VAR
TcUnit.TEST('Test10_CheckIfArrayContainsItem');

ArrayHelper.Clear(arr);
AssertFalse(
	Condition := ArrayHelper.DoesArrayContainItem(arr, item),
	Message := 'Array does not contain the item, method should return FALSE.');

arr[0] := item;

AssertTrue(
	Condition := ArrayHelper.DoesArrayContainItem(arr, item),
	Message := 'Array does contain the item on 0th index, method should return TRUE.');
	
arr[0] := '';
arr[5] := item;

AssertTrue(
	Condition := ArrayHelper.DoesArrayContainItem(arr, item),
	Message := 'Array does contain the item on 5th index, method should return TRUE.');
	
arr[5] := '';
arr[10] := item;	
AssertTrue(
	Condition := ArrayHelper.DoesArrayContainItem(arr, item),
	Message := 'Array does contain the item on 10th index, method should return TRUE.');

arr[0] := 'lalala';
arr[3] := 'aahah';
AssertTrue(
	Condition := ArrayHelper.DoesArrayContainItem(arr, item),
	Message := 'Array does contain the item on 10th index, but also includes non empty elements before, method should return TRUE.');

arr[2] := item;
AssertTrue(
	Condition := ArrayHelper.DoesArrayContainItem(arr, item),
	Message := 'Array does contain the item on 2nd index, but also includes non empty elements before and after, method should return TRUE.');	
	
TcUnit.TEST_FINISHED();
END_METHOD

METHOD Test11_ClearArray_ExpectEmptyArray
VAR_INPUT
END_VAR
VAR_INST
	arrUnmodified	: ARRAY[0..20] OF BOOL;
	arrModified		: ARRAY[0..20] OF BOOL;
	idx				: T_ArrayIndexer;
END_VAR
TcUnit.TEST('Test11_ClearArray_ExpectEmptyArray');

FOR idx := 0 TO 20 BY 1 DO
	arrModified[idx] := TRUE;
END_FOR

AssertTrue(
	Condition := ArrayHelper.Clear(arrModified),
	Message := 'Clearing array returned FALSE when it should have been TRUE.');

AssertArrayEquals_BOOL(
	Actuals := arrModified,
	Expecteds := arrUnmodified,
	Message := 'Array contents were not cleared.');

TcUnit.TEST_FINISHED();
END_METHOD

METHOD Test12_ReferenceToArrayWithAllMethods_ExpectNormalResults
VAR_INST
	arr			: ARRAY[0..10] OF REAL;
	refArr		: REFERENCE TO ARRAY[0..10] OF REAL;
	arrEmpty	: ARRAY[0..10] OF REAL;
	findResult	: REAL;
END_VAR
TcUnit.TEST('Test12_ReferenceToArrayWithAllMethods_ExpectNormalResults');
refarr REF= arr;
arr[5] := 22.2;

ArrayHelper.Clear(refArr);
AssertArrayEquals_REAL(
	Actuals := arr,
	Expecteds := arrEmpty,
	Delta := 0,
	Message := 'Clear array failed.');
	
arr[6] := 5.3;
AssertTrue(
	Condition := ArrayHelper.DoesArrayContainItem(arr := refArr, item := arr[6]),
	Message := 'DoesArrayContainItem failed.');

AssertTrue(
	Condition := ArrayHelper.FindLastOccupiedItem(refArr, refArr[0], findResult),
	Message := 'FindLastOccupiedItem failed (returned FALSE).');

AssertEquals_REAL(
	Actual := findResult,
	Expected := 5.3,
	Delta := 0,
	Message := 'FindLastOccupiedItem output value was incorrect.');
	
AssertEquals_DINT(
	Actual := ArrayHelper.GetElementCount(refArr, refArr[0]),
	Expected := 11,
	Message := 'GetEleeentCount failed.');
	
AssertEquals_DINT(
	Actual := ArrayHelper.GetMaxIndex(refArr, refArr[0], 0),
	Expected := 10,
	Message := 'GetMaxIndex failed.');
	
ArrayHelper.InsertAtStart(refArr, findResult);
AssertEquals_REAL(
	Actual := refArr[0],
	Expected := 5.3,
	Delta := 0.0,
	Message := 'InsertAtStart failed');

arr[0] := 0;	
ArrayHelper.SetAtFirstEmptySlot(refArr, findResult);	
AssertEquals(
	Expected := findResult,
	Actual := refArr[0],
	Message := 'SetAtFirstEmptySlot failed.');
	
arr[1] := 5.5;
ArrayHelper.ShiftDown(refArr, refArr[0]);
AssertEquals_REAL(
	Actual := refArr[0],
	Expected := 5.5,
	Delta := 0.0,
	Message := 'ShiftDown failed.');

ArrayHelper.ShiftUp(refARr, refArr[0]);
AssertEquals_REAL(
	Actual := refArr[1],
	Expected := 5.5,
	Delta := 0.0,
	Message := 'ShiftUp failed.');

TcUnit.TEST_FINISHED();
END_METHOD

METHOD Test13_FindLastOccupiedItem
VAR_INPUT
END_VAR

VAR_INST
	arr	: ARRAY[0..10] OF INT;
	result	: int;
END_VAR
TcUnit.TEST('Test13_FindLastOccupiedItem');

AssertFalse(
	Condition := ArrayHelper.FindLastOccupiedItem(arr, arr[0], result),
	Message := 'Empty array should return FALSE.');
	
arr[5] := 5;

AssertTrue(	
	Condition := ArrayHelper.FindLastOccupiedItem(arr, arr[0], result),
	Message := 'Expected TRUE, 5th element is not empty.');
	
AssertEquals_INT(
	Actual := result,
	Expected := 5,
	Message := 'Incorrect result when finding last occupied element.');
	
TcUnit.TEST_FINISHED();
END_METHOD

METHOD Test14_ShiftDown_ExpectFirstElementOverwriteLastElementZero
VAR_INPUT
END_VAR

VAR
	arr	: ARRAY[0..20] OF INT;
	i	: int;
END_VAR
TcUnit.TEST('Test14_ShiftDown_ExpectFirstElementOverwriteLastElementZero');

FOR i := 0 TO 20 BY 1 DO
	arr[i] := i;
END_FOR

ArrayHelper.ShiftDown(
	arr := arr,
	dataType := arr[0]);
	
AssertEquals_INT(
	Actual := arr[20],
	Expected := 0,
	Message := 'Shifting the array down, last element should be set to 0!');
	
FOR i := 19 TO 0 BY -1 DO
	AssertEquals_INT(
		Actual := arr[i],
		Expected := i+1,
		Message := Tc2_Standard.CONCAT('Shifting up failed! Incorrect value at position ', TO_STRING(i)));
END_FOR
	
TcUnit.TEST_FINISHED();
END_METHOD

END_FUNCTION_BLOCK

// ---- TESTS/Test suites/FB_DateTimeToStringConverter_Tests.TcPOU
FUNCTION_BLOCK INTERNAL FB_DateTimeToStringConverter_Tests EXTENDS FB_TestSuite
VAR_INPUT
END_VAR
VAR_OUTPUT
END_VAR
VAR
	_localSystemTime			: Tc2_Utilities.FB_LocalSystemTime;
	_dateTimeToStringConverter	: FB_DateTimeToStringConverter;
END_VAR

_localSystemTime(
	sNetID:= '', 
	bEnable:= TRUE, 
	dwCycle:= 1);
	
_dateTimeToStringConverter(localSystemTime := _localSystemTime);

Test01_Year();
Test02_Month();
Test03_Day();
Test04_Hour();
Test05_Minute();
Test06_Second();
Test07_Millisecond();

METHOD Test01_Year
VAR_INPUT
END_VAR
TcUnit.TEST('Test01_Year');

AssertEquals_STRING(
	Actual := _dateTimeToStringConverter.Year(),
	Expected := WORD_TO_STRING(_localSystemTime.systemTime.wYear),
	Message := 'Conversion to string for year was incorrect!');
	
TcUnit.TEST_FINISHED();
END_METHOD

METHOD Test02_Month
VAR_INPUT
END_VAR

VAR
	expected	: STRING;
END_VAR
TcUnit.TEST('Test02_Month');

expected := WORD_TO_STRING(_localSystemTime.systemTime.wMonth);

AssertEquals_STRING(
	Actual := _dateTimeToStringConverter.Month(fillWithZeros := FALSE),
	Expected := expected,
	Message := 'Conversion to string for month without zeros was incorrect!');
	
IF LEN(expected) = 1 THEN
	expected := CONCAT('0', WORD_TO_STRING(_localSystemTime.systemTime.wMonth));
END_IF

AssertEquals_STRING(
	Expected := expected,
	Actual := _dateTimeToStringConverter.Month(fillWithZeros := TRUE),
	Message := 'Conversion to string for month with zeros was incorrect!');
	
TcUnit.TEST_FINISHED();
END_METHOD

METHOD PUBLIC Test03_Day

VAR
	expected : STRING;
END_VAR
TcUnit.TEST('Test03_Day');

expected := WORD_TO_STRING(_localSystemTime.systemTime.wDay);

AssertEquals_STRING(
	Actual := _dateTimeToStringConverter.Day(fillWithZeros := FALSE),
	Expected := expected,
	Message := 'Conversion to string for day without zeros was incorrect!');
	
IF LEN(expected) = 1 THEN
	expected := CONCAT('0', WORD_TO_STRING(_localSystemTime.systemTime.wDay));
END_IF

AssertEquals_STRING(
	Expected := expected,
	Actual := _dateTimeToStringConverter.Day(fillWithZeros := TRUE),
	Message := 'Conversion to string for day with zeros was incorrect!');
	
TcUnit.TEST_FINISHED();
END_METHOD

METHOD PUBLIC Test04_Hour

VAR
	expected : STRING;
END_VAR
TcUnit.TEST('Test04_Hour');

expected := WORD_TO_STRING(_localSystemTime.systemTime.wHour);

AssertEquals_STRING(
	Actual := _dateTimeToStringConverter.Hour(fillWithZeros := FALSE),
	Expected := expected,
	Message := 'Conversion to string for hour without zeros was incorrect!');
	
IF LEN(expected) = 1 THEN
	expected := CONCAT('0', WORD_TO_STRING(_localSystemTime.systemTime.wHour));
END_IF

AssertEquals_STRING(
	Expected := expected,
	Actual := _dateTimeToStringConverter.Hour(fillWithZeros := TRUE),
	Message := 'Conversion to string for hour with zeros was incorrect!');
	
TcUnit.TEST_FINISHED();
END_METHOD

METHOD PUBLIC Test05_Minute

VAR
	expected : STRING;
END_VAR
TcUnit.TEST('Test05_Minute');

expected := WORD_TO_STRING(_localSystemTime.systemTime.wMinute);

AssertEquals_STRING(
	Actual := _dateTimeToStringConverter.Minute(fillWithZeros := FALSE),
	Expected := expected,
	Message := 'Conversion to string for minute without zeros was incorrect!');
	
IF LEN(expected) = 1 THEN
	expected := CONCAT('0', WORD_TO_STRING(_localSystemTime.systemTime.wMinute));
END_IF

AssertEquals_STRING(
	Expected := expected,
	Actual := _dateTimeToStringConverter.Minute(fillWithZeros := TRUE),
	Message := 'Conversion to string for minute with zeros was incorrect!');
	
TcUnit.TEST_FINISHED();
END_METHOD

METHOD PUBLIC Test06_Second

VAR
	expected : STRING;
END_VAR
TcUnit.TEST('Test06_Second');

expected := WORD_TO_STRING(_localSystemTime.systemTime.wSecond);

AssertEquals_STRING(
	Actual := _dateTimeToStringConverter.Second(fillWithZeros := FALSE),
	Expected := expected,
	Message := 'Conversion to string for second without zeros was incorrect!');
	
IF LEN(expected) = 1 THEN
	expected := CONCAT('0', WORD_TO_STRING(_localSystemTime.systemTime.wSecond));
END_IF

AssertEquals_STRING(
	Expected := expected,
	Actual := _dateTimeToStringConverter.Second(fillWithZeros := TRUE),
	Message := 'Conversion to string for second with zeros was incorrect!');
	
TcUnit.TEST_FINISHED();
END_METHOD

METHOD PUBLIC Test07_Millisecond

VAR
	expected : STRING;
END_VAR
TcUnit.TEST('Test07_Millisecond');

expected := WORD_TO_STRING(_localSystemTime.systemTime.wMilliseconds);

AssertEquals_STRING(
	Actual := _dateTimeToStringConverter.Millisecond(fillWithZeros := FALSE),
	Expected := expected,
	Message := 'Conversion to string for millisecond without zeros was incorrect!');
	
IF LEN(expected) = 1 THEN
	expected := CONCAT('0', WORD_TO_STRING(_localSystemTime.systemTime.wMilliseconds));
END_IF

AssertEquals_STRING(
	Expected := expected,
	Actual := _dateTimeToStringConverter.Second(fillWithZeros := TRUE),
	Message := 'Conversion to string for millisecond with zeros was incorrect!');
	
TcUnit.TEST_FINISHED();
END_METHOD

END_FUNCTION_BLOCK

// ---- SOURCE/Time/FB_DateTimeToStringConverter.TcPOU
FUNCTION_BLOCK FB_DateTimeToStringConverter IMPLEMENTS I_DateTimeToStringConverter
VAR
	_stringBuilder		: FB_StringBuilder;
END_VAR
VAR_IN_OUT
	localSystemTime	: Tc2_Utilities.FB_LocalSystemTime;
END_VAR

(* Converts TIMESTRUCT to STRING.*)
METHOD DateTime : STRING
VAR_INPUT
	timeFormat			: E_TimeFormat;	// Time format to apply to the timestruct conversion
	timeOfDaySeperator	: STRING(1);	// Specifies how time of day is split
	dateSeperator		: STRING(1);	// Specifies how date is split
	fillWithZeros		: BOOL;	// If set to true: month, day hour, minute and second will have 0 added when only a single digit is present
	IncludeMilliseconds	: BOOL; // If set to true, milliseconds will also be displayed in the result, else they are ignored
END_VAR

VAR
	result			: Tc2_System.T_MaxString;
	stringBuilder	: FB_StringBuilder;
END_VAR
{warning disable C0371}

IF NOT __ISVALIDREF(localSystemTime) THEN
	RETURN;
END_IF

CASE timeFormat OF
	E_TimeFormat.DDMMYY:
		result := stringBuilder.Reset()
			.AddString(THIS^.Day(fillWithZeros))
			.AddString(dateSeperator)
			.AddString(THIS^.Month(fillWithZeros))
			.AddString(dateSeperator)
			.AddString(THIS^.Year())
			.Create();

	E_TimeFormat.HHMMSS:
		result := stringBuilder.Reset()
			.AddString(THIS^.Hour(fillWithZeros))
			.AddString(timeOfDaySeperator)
			.AddString(THIS^.Minute(fillWithZeros))
			.AddString(timeOfDaySeperator)
			.AddString(THIS^.Second(fillWithZeros))
			.Create();
			
		IF IncludeMilliseconds THEN
			result := stringBuilder.AddString(timeOfDaySeperator)
				.AddString(THIS^.Millisecond(fillWithZeros))
				.Create();
		END_IF
			
	E_TimeFormat.MMDDYY:
		result := stringBuilder.Reset()
			.AddString(THIS^.Month(fillWithZeros))
			.AddString(dateSeperator)
			.AddString(THIS^.Day(fillWithZeros))
			.AddString(dateSeperator)
			.AddString(THIS^.Year())
			.Create();

	E_TimeFormat.YYMMDD:	
		result := stringBuilder.Reset()
			.AddString(THIS^.Month(fillWithZeros))
			.AddString(dateSeperator)
			.AddString(THIS^.Day(fillWithZeros))
			.AddString(dateSeperator)
			.AddString(THIS^.Year())
			.Create();
		
	E_TimeFormat.DDMMYY_HHMMSS:
		result := stringBuilder.Reset()
			.AddString(THIS^.Day(fillWithZeros))
			.AddString(dateSeperator)
			.AddString(THIS^.Month(fillWithZeros))
			.AddString(dateSeperator)
			.AddString(THIS^.Year())
			.AddString('_')
			.AddString(THIS^.Hour(fillWithZeros))
			.AddString(timeOfDaySeperator)
			.AddString(THIS^.Minute(fillWithZeros))
			.AddString(timeOfDaySeperator)
			.AddString(THIS^.Second(fillWithZeros))
			.Create();
			
			IF IncludeMilliseconds THEN
				result := stringBuilder.AddString(timeOfDaySeperator)
					.AddString(THIS^.Millisecond(fillWithZeros))
					.Create();
			END_IF

	E_TimeFormat.MMDDYY_HHMMSS:
		result := stringBuilder.Reset()
			.AddString(THIS^.Month(fillWithZeros))
			.AddString(dateSeperator)
			.AddString(THIS^.Day(fillWithZeros))
			.AddString(dateSeperator)
			.AddString(THIS^.Year())
			.AddString('_')
			.AddString(THIS^.Hour(fillWithZeros))
			.AddString(timeOfDaySeperator)
			.AddString(THIS^.Minute(fillWithZeros))
			.AddString(timeOfDaySeperator)
			.AddString(THIS^.Second(fillWithZeros))
			.Create();
			
			IF IncludeMilliseconds THEN
				result := stringBuilder.AddString(timeOfDaySeperator)
					.AddString(THIS^.Millisecond(fillWithZeros))
					.Create();
			END_IF

	E_TimeFormat.YYMMDD_HHMMSS:
		result := stringBuilder.Reset()
			.AddString(THIS^.Year())
			.AddString(dateSeperator)
			.AddString(THIS^.Month(fillWithZeros))
			.AddString(dateSeperator)
			.AddString(THIS^.Day(fillWithZeros))
			.AddString('_')
			.AddString(THIS^.Hour(fillWithZeros))
			.AddString(timeOfDaySeperator)
			.AddString(THIS^.Minute(fillWithZeros))
			.AddString(timeOfDaySeperator)
			.AddString(THIS^.Second(fillWithZeros))
			.Create();
			
			IF IncludeMilliseconds THEN
				result := stringBuilder.AddString(timeOfDaySeperator)
					.AddString(THIS^.Millisecond(fillWithZeros))
					.Create();
			END_IF				
END_CASE

DateTime := result;

{warning restore C0371}
END_METHOD

(* Converts TIMESTRUCT.wDay to STRING.*)
METHOD Day : STRING
VAR_INPUT
	fillWithZeros	: BOOL;	// If set to true, result will have 0 added when only a single digit is present
END_VAR
VAR
	result	: STRING;
END_VAR
{warning disable C0371}

IF NOT __ISVALIDREF(localSystemTime) THEN
	RETURN;
END_IF

result := WORD_TO_STRING(localSystemTime.systemTime.wDay);

IF NOT fillWithZeros THEN
	Day := result;
	RETURN;
END_IF

IF Tc2_Standard.LEN(STR := result) < 2 THEN
	result := Tc2_Standard.CONCAT(STR1 := '0', STR2 := result);
END_IF

Day := result;

{warning restore C0371}
END_METHOD

(* Converts TIMESTRUCT.wHour to STRING.*)
METHOD Hour : STRING
VAR_INPUT
	fillWithZeros	: BOOL;	// If set to true, result will have 0 added when only a single digit is present
END_VAR
VAR
	result	: STRING;
END_VAR
{warning disable C0371}

IF NOT __ISVALIDREF(localSystemTime) THEN
	RETURN;
END_IF

result := WORD_TO_STRING(localSystemTime.systemTime.wHour);

IF NOT fillWithZeros THEN
	Hour := result;
	RETURN;
END_IF

IF Tc2_Standard.LEN(STR := result) < 2 THEN
	result := Tc2_Standard.CONCAT(STR1 := '0', STR2 := result);
END_IF

Hour := result;

{warning restore C0371}
END_METHOD

(* Converts TIMESTRUCT.wMillisecond to STRING.*)
METHOD Millisecond : STRING
VAR_INPUT
	fillWithZeros	: BOOL;	// If set to true, result will have 0 added when only a single digit is present
END_VAR
VAR
	result	: STRING;
END_VAR
{warning disable C0371}

IF NOT __ISVALIDREF(localSystemTime) THEN
	RETURN;
END_IF

result := WORD_TO_STRING(localSystemTime.systemTime.wMilliseconds);

IF NOT fillWithZeros THEN
	Millisecond := result;
	RETURN;
END_IF

IF Tc2_Standard.LEN(STR := result) < 3 THEN
	// _10 => 010
	result := Tc2_Standard.CONCAT(STR1 := '0', STR2 := result);
ELSIF Tc2_Standard.LEN(STR := result) < 2 THEN
	// __5 => 005
	result := Tc2_Standard.CONCAT(STR1 := '00', STR2 := result);
END_IF

Millisecond := result;

{warning restore C0371}
END_METHOD

(* Converts TIMESTRUCT.wMinute to STRING.*)
METHOD Minute : STRING
VAR_INPUT
	fillWithZeros	: BOOL;	// If set to true, result will have 0 added when only a single digit is present
END_VAR
VAR
	result	: STRING;
END_VAR
{warning disable C0371}

IF NOT __ISVALIDREF(localSystemTime) THEN
	RETURN;
END_IF

result := WORD_TO_STRING(localSystemTime.systemTime.wMinute);

IF NOT fillWithZeros THEN
	Minute := result;
	RETURN;
END_IF

IF Tc2_Standard.LEN(STR := result) < 2 THEN
	result := Tc2_Standard.CONCAT(STR1 := '0', STR2 := result);
END_IF

Minute := result;

{warning restore C0371}
END_METHOD

(* Converts TIMESTRUCT.wMonth to STRING.*)
METHOD Month : STRING
VAR_INPUT
	fillWithZeros	: BOOL;	// If set to true, result will have 0 added when only a single digit is present
END_VAR
VAR
	result	: STRING;
END_VAR
{warning disable C0371}

IF NOT __ISVALIDREF(localSystemTime) THEN
	RETURN;
END_IF

result := WORD_TO_STRING(localSystemTime.systemTime.wMonth);

IF NOT fillWithZeros THEN
	Month := result;
	RETURN;
END_IF

IF Tc2_Standard.LEN(STR := result) < 2 THEN
	result := Tc2_Standard.CONCAT(STR1 := '0', STR2 := result);
END_IF

Month := result;

{warning restore C0371}
END_METHOD

(* Converts TIMESTRUCT.wSecond to STRING.*)
METHOD Second : STRING
VAR_INPUT
	fillWithZeros	: BOOL;	// If set to true, result will have 0 added when only a single digit is present
END_VAR
VAR
	result	: STRING;
END_VAR
{warning disable C0371}

IF NOT __ISVALIDREF(localSystemTime) THEN
	RETURN;
END_IF

result := WORD_TO_STRING(localSystemTime.systemTime.wSecond);

IF NOT fillWithZeros THEN
	Second := result;
	RETURN;
END_IF

IF Tc2_Standard.LEN(STR := result) < 2 THEN
	result := Tc2_Standard.CONCAT(STR1 := '0', STR2 := result);
END_IF

Second := result;

{warning restore C0371}
END_METHOD

(* Converts TIMESTRUCT.wYear to STRING.*)
METHOD Year : STRING
VAR
	result	: STRING;
END_VAR
{warning disable C0371}

IF NOT __ISVALIDREF(localSystemTime) THEN
	RETURN;
END_IF

result := WORD_TO_STRING(localSystemTime.systemTime.wYear);
Year := result;

{warning restore C0371}
END_METHOD

END_FUNCTION_BLOCK

// ---- SOURCE/String/StringBuilder/FB_StringBuilder.TcPOU
(* Provides basic string builder implementation.
IMPORTANT NOTE! Doing too many method chains might cause the codesys compiler to either be very slow
when doing the "generating code" part or even fail. Restrain to not using too many or too
many nested methods ( method(fb.Method(fb2.Method())... ).
*)
FUNCTION_BLOCK FB_StringBuilder IMPLEMENTS I_StringBuilder, I_StringBuilderEx_Any 
VAR
	_string	: Tc2_System.T_MaxString;
END_VAR

(* Adds the variable of any data type to the sequence. Conversion is done automatically from within. 
Returns I_StringBuilderEx_Any for further string building capability.

Some extra info: 
	- BOOL and BIT will have the string converted to 'TRUE' and 'FALSE' respectively.
	- BYTE, WORD, DWORD and LWORD will be converted without any additional options. Use AddAnyBit method for these instead!
	- REAL and LREAL will be added as T_MaxString values. Please use AddAnyReal method for these instead.*)

METHOD AddAny : REFERENCE TO FB_StringBuilder
VAR_INPUT
	anyVar	: ANY;
END_VAR

VAR
	result	: Tc2_System.T_MaxString;
	ptrWstring	: POINTER TO WSTRING;
END_VAR
CASE TO_INT(anyVar.TypeClass) OF 
	IBaseLibrary.TypeClass.TYPE_BOOL:
		IF Tc2_Utilities.PBOOL_TO_BOOL(anyVar.pValue) = TRUE THEN
			result :=	'TRUE';
		ELSE
			result := 'FALSE';
		END_IF
		
	IBaseLibrary.TypeClass.TYPE_BYTE: 
		result := BYTE_TO_STRING(Tc2_Utilities.PBYTE_TO_BYTE(anyVar.pValue));
	
	IBaseLibrary.TypeClass.TYPE_DATE:
		result := DATE_TO_STRING(Tc2_Utilities.PDATE_TO_DATE(anyVar.pValue));
	
	IBaseLibrary.TypeClass.TYPE_DATEANDTIME:
		result := DT_TO_STRING(Tc2_Utilities.PDT_TO_DT(anyVar.pValue));
	
	IBaseLibrary.TypeClass.TYPE_DINT:
		result := DINT_TO_STRING(Tc2_Utilities.PDINT_TO_DINT(anyVar.pValue));
	
	IBaseLibrary.TypeClass.TYPE_DWORD:
		result := DWORD_TO_STRING(Tc2_Utilities.PDWORD_TO_DWORD(anyVar.pValue));
	
	IBaseLibrary.TypeClass.TYPE_ENUM:
		result := TO_STRING(anyVar.pValue^);
	
	IBaseLibrary.TypeClass.TYPE_INT:
		result := INT_TO_STRING(Tc2_Utilities.PINT_TO_INT(anyVar.pValue));
	
	IBaseLibrary.TypeClass.TYPE_LINT:
		result := LINT_TO_STRING(Tc2_Utilities.PLINT_TO_LINT(anyVar.pValue));
		
	IBaseLibrary.TypeClass.TYPE_LREAL:
		result := LREAL_TO_STRING(Tc2_Utilities.PLREAL_TO_LREAL(anyVar.pValue));
	
	IBaseLibrary.TypeClass.TYPE_LTIME:
		result := LTIME_TO_STRING(Tc2_Utilities.PLTIME_TO_LTIME(anyVar.pValue));
		
	IBaseLibrary.TypeClass.TYPE_LWORD:
		result := LWORD_TO_STRING(Tc2_Utilities.PLWORD_TO_LWORD(anyVar.pValue));
		
	IBaseLibrary.TypeClass.TYPE_REAL:
		result := REAL_TO_STRING(Tc2_Utilities.PREAL_TO_REAL(anyVar.pValue));
	
	IBaseLibrary.TypeClass.TYPE_SINT:
		result := SINT_TO_STRING(Tc2_Utilities.PSINT_TO_SINT(anyVar.pValue));
	
	IBaseLibrary.TypeClass.TYPE_STRING:
		result := TO_STRING(Tc2_Utilities.PSTRING_TO_STRING(anyVar.pValue));
		
	IBaseLibrary.TypeClass.TYPE_TIME:
		result := TIME_TO_STRING(Tc2_Utilities.PTIME_TO_TIME(anyVar.pValue));
	
	IBaseLibrary.TypeClass.TYPE_TIMEOFDAY:
		result := TOD_TO_STRING(Tc2_Utilities.PTOD_TO_TOD(anyVar.pValue));
	
	IBaseLibrary.TypeClass.TYPE_UDINT:
		result := UDINT_TO_STRING(Tc2_Utilities.PUDINT_TO_UDINT(anyVar.pValue));		
	
	IBaseLibrary.TypeClass.TYPE_UINT:
		result := UINT_TO_STRING(Tc2_Utilities.PUINT_TO_UINT(anyVar.pValue));
	
	IBaseLibrary.TypeClass.TYPE_ULINT:
		result := ULINT_TO_STRING(Tc2_Utilities.PULINT_TO_ULINT(anyVar.pValue));
	
	IBaseLibrary.TypeClass.TYPE_USINT:
		result := USINT_TO_STRING(Tc2_Utilities.PUSINT_TO_USINT(anyVar.pValue));
	
	IBaseLibrary.TypeClass.TYPE_WORD:
		result := WORD_TO_STRING(Tc2_Utilities.PWORD_TO_WORD(anyVar.pValue));
	
	IBaseLibrary.TypeClass.TYPE_WSTRING:
		ptrWstring := anyVar.pValue;
		result := WSTRING_TO_STRING(ptrWstring^);
		
	ELSE
		result := TO_STRING(anyVar.pValue^);
	
END_CASE

THIS^.AddString(result);
AddAny REF= THIS^;
END_METHOD

// Adds a variable of type ANY_BIT to the string generating sequence, based on the provided parameters.
// This includes: BYTE, WORD, DWORD, LWORD, 
METHOD AddAnyBit  : REFERENCE TO FB_StringBuilder
VAR_INPUT
	anyBit					: ANY_BIT;				// Value to be converterd
	option					: E_AddAnyBitOptions;	// Select how the value is converter
	lowerCase				: BOOL;					// If hexadecimal option is selected, the result string can be converted to either lower or upper case
	displayedDigitsCount	: INT;					// This determines how many digits are to be displayed. If actual digits count is lower, the string is filled with zeros from the left side. If left at 0, the result string will be an empty string!
	addNotation				: BOOL;					// If this is set to TRUE, a notation will be prepended: (DEC)10, (BIN)10, (HEX)10, (OCT)10
END_VAR
VAR
	result : Tc2_System.T_MaxString;
END_VAR
CASE anyBit.TypeClass OF
	__SYSTEM.TYPE_CLASS.TYPE_WORD:
		CASE option OF
			E_AddAnyBitOptions.BINARY:
				result := Tc2_Utilities.WORD_TO_BINSTR(
					in := anyBit.pValue^,
					iPrecision := displayedDigitsCount);
				
			E_AddAnyBitOptions.DECIMAL:
				result := Tc2_Utilities.WORD_TO_DECSTR(
					in := anyBit.pValue^,
					iPrecision := displayedDigitsCount);
				
			E_AddAnyBitOptions.HEXADECIMAL:
				result := Tc2_Utilities.WORD_TO_HEXSTR(
					in := anyBit.pValue^,
					iPrecision := displayedDigitsCount,
					bLoCase := lowerCase);
				
			E_AddAnyBitOptions.OCTAL:
				result := Tc2_Utilities.WORD_TO_OCTSTR(
					in := anyBit.pValue^,
					iPrecision := displayedDigitsCount);
		END_CASE
		
	__SYSTEM.TYPE_CLASS.TYPE_BYTE:
		CASE option OF
			E_AddAnyBitOptions.BINARY:
				result := Tc2_Utilities.BYTE_TO_BINSTR(
					in := anyBit.pValue^,
					iPrecision := displayedDigitsCount);
				
			E_AddAnyBitOptions.DECIMAL:
				result := Tc2_Utilities.BYTE_TO_DECSTR(
					in := anyBit.pValue^,
					iPrecision := displayedDigitsCount);
				
			E_AddAnyBitOptions.HEXADECIMAL:
				result := Tc2_Utilities.BYTE_TO_HEXSTR(
					in := anyBit.pValue^,
					iPrecision := displayedDigitsCount,
					bLoCase := lowerCase);
				
			E_AddAnyBitOptions.OCTAL:
				result := Tc2_Utilities.BYTE_TO_OCTSTR(
					in := anyBit.pValue^, 
					iPrecision := displayedDigitsCount);
		END_CASE
	
	__SYSTEM.TYPE_CLASS.TYPE_DWORD:
		CASE option OF
			E_AddAnyBitOptions.BINARY:
				result := Tc2_Utilities.WORD_TO_BINSTR(
					in := anyBit.pValue^,
					iPrecision := displayedDigitsCount);
				
			E_AddAnyBitOptions.DECIMAL:
				result := Tc2_Utilities.WORD_TO_DECSTR(
					in := anyBit.pValue^,
					iPrecision := displayedDigitsCount);
				
			E_AddAnyBitOptions.HEXADECIMAL:
				result := Tc2_Utilities.WORD_TO_HEXSTR(
					in := anyBit.pValue^,
					iPrecision := displayedDigitsCount,
					bLoCase := lowerCase);
				
			E_AddAnyBitOptions.OCTAL:
				result := Tc2_Utilities.WORD_TO_OCTSTR(
					in := anyBit.pValue^,
					iPrecision := displayedDigitsCount);
		END_CASE
	
	__SYSTEM.TYPE_CLASS.TYPE_LWORD:
		CASE option OF
			E_AddAnyBitOptions.BINARY:
				result := Tc2_Utilities.LWORD_TO_BINSTR(
					in := anyBit.pValue^,
					iPrecision := displayedDigitsCount);
				
			E_AddAnyBitOptions.DECIMAL:
				result := Tc2_Utilities.LWORD_TO_DECSTR(
					in := anyBit.pValue^,
					iPrecision := displayedDigitsCount);
				
			E_AddAnyBitOptions.HEXADECIMAL:
				result := Tc2_Utilities.LWORD_TO_HEXSTR(
					in := anyBit.pValue^,
					iPrecision := displayedDigitsCount,
					bLoCase := lowerCase);
				
			E_AddAnyBitOptions.OCTAL:
				result := Tc2_Utilities.LWORD_TO_OCTSTR(
					in := anyBit.pValue^,
					iPrecision := displayedDigitsCount);
		END_CASE
END_CASE

IF addNotation THEN
	CASE option OF
		E_AddAnyBitOptions.BINARY:
			result := Tc2_Standard.CONCAT('(BIN)', result);
			
		E_AddAnyBitOptions.DECIMAL:
			result := Tc2_Standard.CONCAT('(DEC)', result);
		
		E_AddAnyBitOptions.HEXADECIMAL:
			result := Tc2_Standard.CONCAT('(HEX)', result);
		
		E_AddAnyBitOptions.OCTAL:
			result := Tc2_Standard.CONCAT('(OCT)', result);
	END_CASE
END_IF

THIS^.AddString(result);
AddAnyBit REF= THIS^;
END_METHOD

// Adds any REAL or LREAL value to the generating string sequence.
// Please note that REAL values will ALWAYS be automatically rounded on 3rd decimal digit.
// Anything after it will be whatever TwinCAT decides to do.
METHOD AddAnyReal : REFERENCE TO FB_StringBuilder
VAR_INPUT
	anyReal		: ANY_REAL;	// Value to be converter
	precision	: INT;		// Precision of decimal digits
	round		: BOOL;		// Rounding of the last displayed digit
END_VAR
IF anyReal.diSize = SIZEOF(REAL) THEN
	// REAL
	THIS^.AddString(
		Tc2_Utilities.LREAL_TO_FMTSTR(
			in := REAL_TO_LREAL(Tc2_Utilities.PREAL_TO_REAL(anyReal.pValue)),
			iPrecision := precision, 
			bRound := round));
		
ELSE
	// LREAL
	THIS^.AddString(Tc2_Utilities.LREAL_TO_FMTSTR(
		in := Tc2_Utilities.PLREAL_TO_LREAL(anyReal.pValue),
		iPrecision := precision,
		bRound := round));	
END_IF

AddAnyReal REF= THIS^;
END_METHOD

(* Adds a string to the build sequence.*)
METHOD AddString : REFERENCE TO FB_StringBuilder
VAR_INPUT
	(* String to be added.*)
	str	: Tc2_System.T_MaxString;
END_VAR
_string := Tc2_Standard.CONCAT(
	STR1 := _string, 
	STR2 := str);
	
AddString  REF= THIS^;
END_METHOD

(* Adds a string to the build sequence and wraps the str in double quotation marks "str"*)
METHOD AddWithDblQuotationMarks : REFERENCE TO FB_StringBuilder
VAR_INPUT
	str	: Tc2_System.T_MaxString;
END_VAR
_string := Tc2_Standard.CONCAT(
	STR1 := _string, 
	STR2 := Tc2_Standard.CONCAT(
		STR1 := StringConstants.DoubleQuotationMark, 
		STR2 := Tc2_Standard.CONCAT(
			STR1 := str, 
			STR2 := StringConstants.DoubleQuotationMark))); 
	
AddWithDblQuotationMarks  REF= THIS^;
END_METHOD

(* Adds a string to the build sequence and wraps the str in quotation marks 'str'*)
METHOD AddWithQuotationMark : REFERENCE TO FB_StringBuilder
VAR_INPUT
	str	: Tc2_System.T_MaxString;
END_VAR
_string := Tc2_Standard.CONCAT(
	STR1 := _string, 
	STR2 := Tc2_Standard.CONCAT(
		STR1 := StringConstants.SingleQuotationMark, 
		STR2 := Tc2_Standard.CONCAT(
			STR1 := str, 
			STR2 := StringConstants.SingleQuotationMark))); 
		
AddWithQuotationMark REF= THIS^;
END_METHOD

(* Finishes string generation and returns the generated string*)
METHOD Create : Tc2_System.T_MaxString
Create := _string;
END_METHOD

(* Reset the string build sequence, clear any string built so far.*)
METHOD Reset : REFERENCE TO FB_StringBuilder
_string := '';
Reset REF= THIS^;
END_METHOD

END_FUNCTION_BLOCK

// ---- SOURCE/String/StringConstants.TcPOU
(* Contains string constants
A STRING constant is a string enclosed by single quotation marks. The characters are encoded according to the Windows 1252 character set. 
As a subset of Windows-1252, the character set of ISO/IEC 8859-1 is supported. 
A STRING constant can contain blanks and umlauts, since these characters are part of the character set. 
It is also referred to as a character literal or simply a string.*)

PROGRAM StringConstants
VAR CONSTANT
	LineFeed			: STRING := '$L';
	NewLine				: STRING := '$N';
	FormFeed			: STRING := '$P';
	LineBreak			: STRING := '$R';
	Tab					: STRING := '$T';
	DollarSign			: STRING := '$$';
	SingleQuotationMark	: STRING := '$'';
	DoubleQuotationMark	: STRING := '$22';
END_VAR

END_PROGRAM

// ---- TESTS/Test suites/FB_ErrorSource_Tests.TcPOU
FUNCTION_BLOCK INTERNAL FB_ErrorSource_Tests EXTENDS FB_TestSuite
VAR_INPUT
END_VAR
VAR_OUTPUT
END_VAR
VAR
	_errorSourceObject	: FB_ErrorSource_ExtensionForTests;
END_VAR

Test01_ErrorProperty();
Test02_ErrorCode();
Test03_ErrorMessage();
Test04_GenericError();

METHOD Test01_ErrorProperty
VAR_INPUT
END_VAR
TcUnit.TEST('Test01_ErrorProperty');
_errorSourceObject.bError := TRUE;
_errorSourceObject();
AssertTrue(
	Condition := _errorSourceObject.Error,
	Message := 'Error should be TRUE.');	
	
TcUnit.TEST_FINISHED();
END_METHOD

METHOD Test02_ErrorCode
VAR
END_VAR
TcUnit.TEST('Test02_ErrorCode');

_errorSourceObject.eAdsErrorCodeToTest := TcError.AdsErrorCodes.ADSERR_CLIENT_ERROR;
_errorSourceObject();

AssertEquals_UDINT(
	Actual := _errorSourceObject.AdsError.Code,
	Expected := TcError.AdsErrorCodes.ADSERR_CLIENT_ERROR,
	Message := 'The error code provided in the ErrorInfo.Code property is incorrect!');

TcUnit.TEST_FINISHED();
END_METHOD

METHOD PRIVATE Test03_ErrorMessage
VAR_INPUT
END_VAR
TcUnit.TEST('Test03_ErrorMessage');

_errorSourceObject.eAdsErrorCodeToTest := TcError.AdsErrorCodes.ADSERR_DEVICE_ABORTED;
_errorSourceObject();

AssertEquals_STRING(
	Actual := _errorSourceObject.AdsError.Message,
	Expected := 'Request is aborted.',
	Message := 'The error information was incorrect!');

TcUnit.TEST_FINISHED();
END_METHOD

METHOD Test04_GenericError
VAR_INPUT
END_VAR
TcUnit.TEST('Test04_GenericError');

_errorSourceObject.nGenericErrorCode := 10;
_errorSourceObject.sGenericErrorMessage := 'Error message, generic...';
_errorSourceObject();
AssertEquals_DINT(
	Expected := 10,
	Actual := _errorSourceObject.GenericError.Code,
	Message := 'Incorrect error code.');
	
AssertEquals_STRING(
	Expected := 'Error message, generic...',
	Actual := _errorSourceObject.GenericError.Message,
	Message := 'Incorrect error message.');
	
TcUnit.TEST_FINISHED();
END_METHOD

END_FUNCTION_BLOCK

// ---- TESTS/Test suites/FB_ErrorSource_ExtensionForTests.TcPOU
// Since FB_ErrorSource is an ABSTRACT class, the functionality needs to be implemented by extending the base class
FUNCTION_BLOCK INTERNAL FB_ErrorSource_ExtensionForTests EXTENDS FB_ErrorSource
VAR_INPUT
	eAdsErrorCodeToTest 	: TcError.AdsErrorCodes;
	sGenericErrorMessage	: Tc2_System.T_MaxString;
	nGenericErrorCode		: DINT;
	bError					: BOOL;		
END_VAR

THIS^.AdsError.Code := eAdsErrorCodeToTest;
THIS^.GenericError.Message := sGenericErrorMessage;
THIS^.GenericError.Code := nGenericErrorCode;
THIS^.Error := bError;

END_FUNCTION_BLOCK

// ---- SOURCE/Errors/FB_ErrorSource.TcPOU
// Provides I_ErrorSource base implementation.

{attribute 'no_explicit_call' := 'Body contains no logic, calling methods only allowed.'}
FUNCTION_BLOCK ABSTRACT FB_ErrorSource EXTENDS FB_HasInstanceNameAndPath IMPLEMENTS I_ErrorSource
VAR
	_adsError		: ST_AdsError;
	_error			: BOOL;
	_genericError	: ST_GenericError;
END_VAR

// Gets or sets the Ads error - note that code to message conversion is done automatically.
{attribute 'monitoring':='call'}
PROPERTY AdsError : REFERENCE TO ST_AdsError
GET
_adsError.Message := TcError.AdsErrorCodeDescription(_adsError.Code);
AdsError REF= _adsError;
END_GET
SET // PROTECTED
_adsError := AdsError;
END_SET
END_PROPERTY

{attribute 'monitoring':='call'}
(* Returns TRUE if an error has occurred*)
PROPERTY Error : BOOL
GET
Error := _error;
END_GET
SET // PROTECTED
_error := Error;
END_SET
END_PROPERTY

{attribute 'monitoring':='call'}
PROPERTY GenericError : REFERENCE TO ST_GenericError
GET
GenericError REF= _genericError;
END_GET
SET // PROTECTED
_genericError := GenericError;
END_SET
END_PROPERTY

// Reset all errors
METHOD PROTECTED ResetError : BOOL
VAR_INPUT
END_VAR
THIS^.Error := FALSE;
THIS^.AdsError.Code := TcError.ToAdsErrorCode(0);
THIS^.AdsError.Source := '';
THIS^.GenericError.Code := 0;
THIS^.GenericError.Source := '';
END_METHOD

END_FUNCTION_BLOCK

// ---- SOURCE/General/FB_HasInstanceNameAndPath.TcPOU
// When inherited, the child function block will gain two properties:
// InstanceName - ONLY the name of the instantiated function block
// InstancePath - the FULL instance path

{attribute 'reflection'}
{attribute 'hide_all_locals'}
{attribute 'no_explicit_call' := 'Body contains no logic, calling methods only allowed.'}
FUNCTION_BLOCK ABSTRACT FB_HasInstanceNameAndPath
VAR
	{attribute 'instance-path'} 
    {attribute 'noinit'} 
	_instancePath	: Tc2_System.T_MaxString;
	_instanceName	: Tc2_System.T_MaxString;
END_VAR

{attribute 'hide'}
METHOD FB_init : BOOL
VAR_INPUT
	bInitRetains : BOOL; // if TRUE, the retain variables are initialized (warm start / cold start)
	bInCopyCode : BOOL;  // if TRUE, the instance afterwards gets moved into the copy code (online change)
END_VAR
_instanceName := InstanceNameHelper.InstanceNameFromPath(_instancePath, 10);
_instancePath := InstanceNameHelper.RemoveProjectFromInstancePath(_instancePath);
END_METHOD

{attribute 'monitoring':='call'}
PROPERTY InstanceName : Tc2_System.T_MaxString
GET
InstanceName := _instanceName;
END_GET
END_PROPERTY

{attribute 'monitoring':='call'}
PROPERTY InstancePath : Tc2_System.T_MaxString
GET
VAR
	varInfo	: T_VarInfo;
END_VAR
InstancePath := _instancePath;
END_GET
END_PROPERTY

END_FUNCTION_BLOCK

// ---- SOURCE/General/InstanceNameHelper.TcPOU
PROGRAM InstanceNameHelper
VAR
END_VAR

METHOD InstanceNameFromPath : T_MaxString
VAR_INPUT
	path		: Tc2_System.T_MaxString;
	maxAttempts	: INT;
END_VAR
VAR
	instanceName	: Tc2_System.T_MaxString;
	dotPosition		: INT;
	iteration		: INT;
	
END_VAR

VAR CONSTANT
	ABSOLUTE_MAX_ATTEMPTS : INT := 20;
END_VAR
instanceName := path;

// Limiting maximum number of dots in the instancePath to maximum of 20 with ABSOLUTE_MAX_ATTEMPTS
// This is mostly important due to the method being called in FB_Init, where I think too long method calls shouldn't be happening.
// In theory, I don't think it would ever go above 10, unless some very deep object nesting is done.
// Example Project.Plc.Main.Fb.Fb.Fb.Fb.Fb...

WHILE Tc2_Standard.FIND(STR1 := instanceName, STR2 := '.') <> 0 AND 
	 (iteration < MIN(maxAttempts, ABSOLUTE_MAX_ATTEMPTS)) 
DO
	dotPosition := Tc2_Standard.FIND(
		STR1 := instanceName, 
		STR2 := '.');
		
	instanceName := Tc2_Standard.DELETE(
		STR := instanceName,
		POS := 1,	
		LEN := dotPosition);
		
	iteration := iteration + 1;
END_WHILE

InstanceNameFromPath := instanceName;
END_METHOD

METHOD RemoveProjectFromInstancePath : T_MaxString
VAR_INPUT
	instancePath	: Tc2_System.T_MaxString;
END_VAR
VAR
	result		: Tc2_System.T_MaxString;
	dotPosition	: INT;
	iteration	: INT;
END_VAR

VAR CONSTANT
	FILE_PREIX_DOTS_TO_REMOVE	: INT := 2;
END_VAR
RemoveProjectFromInstancePath := InstanceNameFromPath(instancePath,2);
END_METHOD

END_PROGRAM

// ---- TESTS/Test suites/FB_HasInstanceName_Tests.TcPOU
FUNCTION_BLOCK INTERNAL FB_HasInstanceName_Tests EXTENDS FB_TestSuite
VAR_INPUT
END_VAR
VAR_OUTPUT
END_VAR
VAR
	fbHasInstanceName	:  FB_HasInstanceName_ExtensionForTests;
END_VAR

Test01_InstanceName();
Test02_InstancePath();

METHOD Test01_InstanceName
VAR_INPUT
END_VAR
TcUnit.TEST('Test01_InstanceName');

AssertEquals_STRING(
	Expected := 'fbHasInstanceName',
	Actual := fbHasInstanceName.InstanceName,
	Message := 'InstanceName is not correct.');
	
TcUnit.TEST_FINISHED();
END_METHOD

METHOD Test02_InstancePath
VAR_INPUT
END_VAR
TcUnit.TEST('Test02_InstancePath');

AssertEquals_STRING(
	Expected := 'PRG_TESTS.HasInstanceNameTests.fbHasInstanceName',
	Actual := fbHasInstanceName.InstancePath,
	Message := 'Instance path is incorrect.');

TcUnit.TEST_FINISHED();
END_METHOD

END_FUNCTION_BLOCK

// ---- TESTS/Test suites/FB_HasInstanceName_ExtensionForTests.TcPOU
// Since FB_HasInstanceName is an ABSTRACT class, 
// the functionality needs to be implemented by extending the base class
FUNCTION_BLOCK INTERNAL FB_HasInstanceName_ExtensionForTests EXTENDS FB_HasInstanceNameAndPath
VAR_INPUT
END_VAR
VAR_OUTPUT
END_VAR
VAR
END_VAR

END_FUNCTION_BLOCK

// ---- TESTS/Test suites/FB_StringBuilder_Tests.TcPOU
FUNCTION_BLOCK INTERNAL FB_StringBuilder_Tests EXTENDS FB_StringBuilderEx_Any_Tests
VAR_INPUT
END_VAR
VAR_OUTPUT
END_VAR
VAR
	_stringBuilder	: FB_StringBuilder;
END_VAR

Test01_AddStrings_ExpectConcat();
Test02_AddWithSingleQuotationMarks();
Test03_AddWithDoubleQuotationMarks();
Test04_CreateDoesNotResetStringSequence();
Test05_ResetClearsBuildSequence();
SUPER^();

METHOD Test01_AddStrings_ExpectConcat
VAR_INPUT
END_VAR
IF TcUnit.TEST_ORDERED('Test01_AddStrings_ExpectConcat') THEN
	AssertEquals_STRING(
		Actual := _stringBuilder.Reset()
			.AddString('test')
			.AddString('test2')
			.Create(),
		Expected := 'testtest2',
		Message := 'AddString of two strings failed!');
		
	TcUnit.TEST_FINISHED();
END_IF
END_METHOD

METHOD Test02_AddWithSingleQuotationMarks
VAR_INPUT
END_VAR
IF TcUnit.TEST_ORDERED('Test02_AddWithSingleQuotationMarks') THEN
	AssertEquals_STRING(
		Actual := _stringBuilder.Reset()
			.AddWithQuotationMark('test')
			.AddWithQuotationMark('test2')
			.Create(),
		Expected := '$'test$'$'test2$'',
		Message := 'AddString of two strings failed!');
		
	TcUnit.TEST_FINISHED();
END_IF
END_METHOD

METHOD Test03_AddWithDoubleQuotationMarks
VAR_INPUT
END_VAR
IF TcUnit.TEST_ORDERED('Test03_AddWithDoubleQuotationMarks') THEN
	AssertEquals_STRING(
		Actual := _stringBuilder.Reset()
			.AddWithDblQuotationMarks('test')
			.AddWithDblQuotationMarks('test2')
			.Create(),
		Expected := '"test""test2"',
		Message := 'AddString of two strings failed!');
		
	TcUnit.TEST_FINISHED();
END_IF
END_METHOD

METHOD Test04_CreateDoesNotResetStringSequence
VAR_INPUT
END_VAR
IF TcUnit.TEST_ORDERED('Test04_CreateDoesNotResetStringSequence') THEN
	_stringBuilder.Reset()
		.AddString('a')
		.AddString('b')
		.Create();
		
	AssertEquals_STRING(
		Actual := _stringBuilder.AddString('c').Create(),
		Expected := 'abc',
		Message := 'Calling .Create() should result in the string creation remaining intact, until Reset() is called explicitly!');
		
	TcUnit.TEST_FINISHED();
END_IF
END_METHOD

METHOD Test05_ResetClearsBuildSequence
VAR_INPUT
END_VAR
IF TcUnit.TEST_ORDERED('Test05_ResetClearsBuildSequence') THEN
	_stringBuilder.Reset()
		.AddString('a')
		.AddString('b')
		.Reset()
		.AddString('c');
	
	AssertEquals_STRING(
		Actual := _stringBuilder.Create(),
		Expected := 'c',
		Message := 'Calling Reset() method should result in the sequnce being cleared!');
		
	TcUnit.TEST_FINISHED();
END_IF
END_METHOD

END_FUNCTION_BLOCK

// ---- TESTS/Test suites/FB_StringBuilderEx_Any_Tests.TcPOU
FUNCTION_BLOCK INTERNAL FB_StringBuilderEx_Any_Tests EXTENDS TcUnit.FB_TestSuite
VAR_INPUT
END_VAR
VAR_OUTPUT
END_VAR
VAR
	stringBuilder	: FB_StringBuilder;
END_VAR

Test01_BOOL();
Test02_BYTE();
Test03_DATE();
Test04_DateAndTime();
Test05_DINT();
Test06_DWORD();
Test07_ENUM();
Test08_INT();
Test09_LINT();
Test10_LREAL();
Test11_LTIME();
Test12_LWORD();
Test13_REAL();
Test14_SINT();
Test15_STRING();
Test16_TIME();
Test17_TOD();
Test18_UDINT();
Test19_UINT();
Test20_ULINT();
Test21_USINT();
Test22_WORD();
Test23_WSTRING();
Test24_ANY_BIT_WORD();
Test25_ANY_BIT_BYTE();
Test26_ANY_BIT_DWORD();
Test27_ANY_BIT_LWORD();
Test28_ANY_REAL_REAL();
Test29_ANY_REAL_LREAL();

METHOD Test01_BOOL
VAR_INPUT
END_VAR

VAR_INST
	bTrue		: BOOL := TRUE;
	bFalse		: BOOL := FALSE;

END_VAR
IF TcUnit.TEST_ORDERED('Test01_BOOL') THEN
	AssertEquals_STRING(
		Actual := stringBuilder.Reset().AddAny(bTrue).Create(),
		Expected := 'TRUE',
		Message := 'Adding boolean failed');
		
	AssertEquals_STRING(
		Actual := stringBuilder.Reset().AddAny(bFalse).Create(),
		Expected := 'FALSE',
		Message := 'Adding boolean failed');
		
	TcUnit.TEST_FINISHED();
END_IF
END_METHOD

METHOD Test02_BYTE
VAR_INPUT
END_VAR
VAR
	byteVar	: BYTE := 17;
END_VAR
IF TEST_ORDERED('Test02_BYTE') THEN
	
	AssertEquals_STRING(
		Actual := stringBuilder.Reset().AddAny(byteVar).Create(),
		Expected := '17',
		Message := 'Adding BYTE failed.');
	TEST_FINISHED();
END_IF
END_METHOD

METHOD Test03_DATE
VAR
	someVar	: DATE := D#1970-01-01;
END_VAR
IF TEST_ORDERED('Test03_DATE') THEN
	AssertEquals_STRING(
		Actual := stringBuilder.Reset().AddAny(someVar).Create(),
		Expected := 'D#1970-01-01',
		Message := 'Adding DATE failed.');

	TEST_FINISHED();
END_IF
END_METHOD

METHOD Test04_DateAndTime
VAR
	someVar	: DATE_AND_TIME := DT#1970-1-1-0:0:1;
END_VAR
IF TEST_ORDERED('Test04_DateAndTime') THEN
	AssertEquals_STRING(
		Actual := stringBuilder.Reset().AddAny(someVar).Create(),
		Expected := 'DT#1970-01-01-00:00:01',
		Message := 'Adding DATE_AND_TIME failed.');

	TEST_FINISHED();
END_IF
END_METHOD

METHOD Test05_DINT
VAR
	someVar	: DINT := 15;
END_VAR
IF TEST_ORDERED('Test05_DINT') THEN
	AssertEquals_STRING(
		Actual := stringBuilder.Reset().AddAny(someVar).Create(),
		Expected := '15',
		Message := 'Adding DINT failed.');

	TEST_FINISHED();
END_IF
END_METHOD

METHOD Test06_DWORD
VAR
	someVar	: DWORD := 777;
END_VAR
IF TEST_ORDERED('Test06_DWORD') THEN
	AssertEquals_STRING(
		Actual := stringBuilder.Reset().AddAny(someVar).Create(),
		Expected := '777',
		Message := 'Adding DWORD failed.');

	TEST_FINISHED();
END_IF
END_METHOD

METHOD Test07_ENUM
VAR
	someVar	: E_AddAnyBitOptions := E_AddAnyBitOptions.HEXADECIMAL;
END_VAR
IF TEST_ORDERED('Test07_ENUM') THEN
	AssertEquals_STRING(
		Actual := stringBuilder.Reset().AddAny(someVar).Create(),
		Expected := '2',
		Message := 'Adding ENUM failed.');

	TEST_FINISHED();
END_IF
END_METHOD

METHOD Test08_INT
VAR
	someVar	: INT := 22;
END_VAR
IF TEST_ORDERED('Test08_INT') THEN
	AssertEquals_STRING(
		Actual := stringBuilder.Reset().AddAny(someVar).Create(),
		Expected := '22',
		Message := 'Adding INT failed.');

	TEST_FINISHED();
END_IF
END_METHOD

METHOD Test09_LINT
VAR
	someVar	: LINT := 6666;
END_VAR
IF TEST_ORDERED('Test09_LINT') THEN
	AssertEquals_STRING(
		Actual := stringBuilder.Reset().AddAny(someVar).Create(),
		Expected := '6666',
		Message := 'Adding LINT failed.');

	TEST_FINISHED();
END_IF
END_METHOD

METHOD Test10_LREAL
VAR
	someVar	: LREAL := 11.11;
END_VAR
IF TEST_ORDERED('Test10_LREAL') THEN
	AssertEquals_STRING(
		Actual := stringBuilder.Reset().AddAny(someVar).Create(),
		Expected := '11.11',
		Message := 'Adding LREAL failed.');

	TEST_FINISHED();
END_IF
END_METHOD

METHOD Test11_LTIME
VAR
	someVar	: LTIME := LTIME#100D2H30M40S500MS600US700NS;
END_VAR
IF TEST_ORDERED('Test11_LTIME') THEN
	AssertEquals_STRING(
		Actual := stringBuilder.Reset().AddAny(someVar).Create(),
		Expected := 'LTIME#100d2h30m40s500ms600us700ns',
		Message := 'Adding LTIME failed.');

	TEST_FINISHED();
END_IF
END_METHOD

METHOD Test12_LWORD
VAR
	someVar	: LWORD := 123456;
END_VAR
IF TEST_ORDERED('Test12_LWORD') THEN
	AssertEquals_STRING(
		Actual := stringBuilder.Reset().AddAny(someVar).Create(),
		Expected := '123456',
		Message := 'Adding LWORD failed.');

	TEST_FINISHED();
END_IF
END_METHOD

METHOD Test13_REAL
VAR
	someVar	: REAL := 12345.6789;
END_VAR
IF TEST_ORDERED('Test13_REAL') THEN
	AssertEquals_STRING(
		Actual := stringBuilder.Reset().AddAny(someVar).Create(),
		Expected := '12345.679',
		Message := 'Adding REAL failed.');

	TEST_FINISHED();
END_IF
END_METHOD

METHOD Test14_SINT
VAR
	someVar	: SINT := -34;
END_VAR
IF TEST_ORDERED('Test14_SINT') THEN
	AssertEquals_STRING(
		Actual := stringBuilder.Reset().AddAny(someVar).Create(),
		Expected := '-34',
		Message := 'Adding SINT failed.');

	TEST_FINISHED();
END_IF
END_METHOD

METHOD Test15_STRING
VAR
	someVar	: STRING := 'haha';
END_VAR
IF TEST_ORDERED('Test15_STRING') THEN
	AssertEquals_STRING(
		Actual := stringBuilder.Reset().AddAny(someVar).Create(),
		Expected := 'haha',
		Message := 'Adding STRING failed.');

	TEST_FINISHED();
END_IF
END_METHOD

METHOD Test16_TIME
VAR
	someVar	: TIME := T#15D10S;
END_VAR
IF TEST_ORDERED('Test16_TIME') THEN
	AssertEquals_STRING(
		Actual := stringBuilder.Reset().AddAny(someVar).Create(),
		Expected := 'T#15d10s',
		Message := 'Adding TIME failed.');

	TEST_FINISHED();
END_IF
END_METHOD

METHOD Test17_TOD
VAR
	someVar	: TOD := TOD#14:01:05.123;
END_VAR
IF TEST_ORDERED('Test17_TOD') THEN
	AssertEquals_STRING(
		Actual := stringBuilder.Reset().AddAny(someVar).Create(),
		Expected := 'TOD#14:01:05.123',
		Message := 'Adding TOD failed.');

	TEST_FINISHED();
END_IF
END_METHOD

METHOD Test18_UDINT
VAR
	someVar	: UDINT := 23452352;
END_VAR
IF TEST_ORDERED('Test18_UDINT') THEN
	AssertEquals_STRING(
		Actual := stringBuilder.Reset().AddAny(someVar).Create(),
		Expected := '23452352',
		Message := 'Adding UDINT failed.');

	TEST_FINISHED();
END_IF
END_METHOD

METHOD Test19_UINT
VAR
	someVar	: UINT := 12341;
END_VAR
IF TEST_ORDERED('Test19_UINT') THEN
	AssertEquals_STRING(
		Actual := stringBuilder.Reset().AddAny(someVar).Create(),
		Expected := '12341',
		Message := 'Adding UINT failed.');

	TEST_FINISHED();
END_IF
END_METHOD

METHOD Test20_ULINT
VAR
	someVar	: ULINT := 12345678;
END_VAR
IF TEST_ORDERED('Test20_ULINT') THEN
	AssertEquals_STRING(
		Actual := stringBuilder.Reset().AddAny(someVar).Create(),
		Expected := '12345678',
		Message := 'Adding ULINT failed.');

	TEST_FINISHED();
END_IF
END_METHOD

METHOD Test21_USINT
VAR
	someVar	: USINT := 123;
END_VAR
IF TEST_ORDERED('Test21_USINT') THEN
	AssertEquals_STRING(
		Actual := stringBuilder.Reset().AddAny(someVar).Create(),
		Expected := '123',
		Message := 'Adding USINT failed.');

	TEST_FINISHED();
END_IF
END_METHOD

METHOD Test22_WORD
VAR
	someVar	: WORD := 16#A;
END_VAR
IF TEST_ORDERED('Test22_WORD') THEN
	AssertEquals_STRING(
		Actual := stringBuilder.Reset().AddAny(someVar).Create(),
		Expected := '10',
		Message := 'Adding WORD failed.');

	TEST_FINISHED();
END_IF
END_METHOD

METHOD Test23_WSTRING
VAR
	someVar	: WSTRING := "test";
END_VAR
IF TEST_ORDERED('Test23_WSTRING') THEN
	AssertEquals_STRING(
		Actual := stringBuilder.Reset().AddAny(someVar).Create(),
		Expected := 'test',
		Message := 'Adding WSTRING failed.');

	TEST_FINISHED();
END_IF
END_METHOD

METHOD Test24_ANY_BIT_WORD
VAR_INPUT
END_VAR
VAR
	wordVar	: WORD := 16#AB;
	result	: Tc2_System.T_MaxString;
END_VAR
IF TcUnit.TEST_ORDERED('Test24_ANY_BIT_WORD') THEN
	
	// BINARY with notations
	result := stringBuilder.Reset().
		AddAnyBit(
			anyBit := wordVar, 
			option := E_AddAnyBitOptions.BINARY, 
			lowerCase := FALSE, 
			displayedDigitsCount := 16, 
			addNotation := TRUE)
		.Create();
		
	AssertEquals_STRING(
		Actual := result,
		Expected := '(BIN)0000000010101011',
		Message := 'Adding word as BINARY with addNotation = TRUE was incorrect');
		
	// BINARY without notations
	result := stringBuilder.Reset()
		.AddAnyBit(
			anyBit := wordVar, 
			option := E_AddAnyBitOptions.BINARY, 
			lowerCase := FALSE, 
			displayedDigitsCount := 16, 
			addNotation := FALSE)
		.Create();
		
	AssertEquals_STRING(
		Actual := result,
		Expected := '0000000010101011',
		Message := 'Adding word as BINARY with addNotation = FALSE was incorrect');
		
	// DECIMAL with notations
	result := stringBuilder.Reset()
		.AddAnyBit(
			anyBit := wordVar, 
			option := E_AddAnyBitOptions.DECIMAL, 
			lowerCase := FALSE, 
			displayedDigitsCount := 16, 
			addNotation := TRUE)
		.Create();
		
	AssertEquals_STRING(
		Actual := result,
		Expected := '(DEC)0000000000000171',
		Message := 'Adding word as DECIMAL with addNotation = TRUE was incorrect');
		
	// DECIMAL without notations
	result := stringBuilder.Reset()
		.AddAnyBit(
			anyBit := wordVar, 
			option := E_AddAnyBitOptions.DECIMAL, 
			lowerCase := FALSE, 
			displayedDigitsCount := 16, 
			addNotation := FALSE)
		.Create();
		
	AssertEquals_STRING(
		Actual := result,
		Expected := '0000000000000171',
		Message := 'Adding word as DECIMAL with addNotation = FALSE was incorrect');

	// HEXADECIMAL with notations
	result := stringBuilder.Reset()
		.AddAnyBit(
			anyBit := wordVar, 
			option := E_AddAnyBitOptions.HEXADECIMAL, 
			lowerCase := FALSE, 
			displayedDigitsCount := 16, 
			addNotation := TRUE)
		.Create();
		
	AssertEquals_STRING(
		Actual := result,
		Expected := '(HEX)00000000000000AB',
		Message := 'Adding word as HEXADECIMAL with addNotation = TRUE was incorrect');
		
	// HEXADECIMAL without notations
	result := stringBuilder.Reset()
		.AddAnyBit(
			anyBit := wordVar, 
			option := E_AddAnyBitOptions.HEXADECIMAL, 
			lowerCase := FALSE, 
			displayedDigitsCount := 16, 
			addNotation := FALSE)
		.Create();
		
	AssertEquals_STRING(
		Actual := result,
		Expected := '00000000000000AB',
		Message := 'Adding word as HEXADECIMAL with addNotation = FALSE was incorrect');
	
	// OCTAL with notations
	result := stringBuilder.Reset()
		.AddAnyBit(
			anyBit := wordVar, 
			option := E_AddAnyBitOptions.OCTAL, 
			lowerCase := FALSE, 
			displayedDigitsCount := 16, 
			addNotation := TRUE)
		.Create();
		
	AssertEquals_STRING(
		Actual := result,
		Expected := '(OCT)0000000000000253',
		Message := 'Adding word as OCTAL with addNotation = TRUE was incorrect');
		
	// OCTAL without notations
	result := stringBuilder.Reset()
		.AddAnyBit(
			anyBit := wordVar, 
			option := E_AddAnyBitOptions.OCTAL, 
			lowerCase := FALSE, 
			displayedDigitsCount := 16, 
			addNotation := FALSE)
		.Create();
		
	AssertEquals_STRING(
		Actual := result,
		Expected := '0000000000000253',
		Message := 'Adding word as OCTAL with addNotation = FALSE was incorrect');
		
	TcUnit.TEST_FINISHED();
END_IF
END_METHOD

METHOD Test25_ANY_BIT_BYTE
VAR_INPUT
END_VAR
VAR
	byteVar	: BYTE := 16#AB;
	result	: Tc2_System.T_MaxString;
END_VAR
IF TcUnit.TEST_ORDERED('Test25_ANY_BIT_BYTE') THEN
	
	// BINARY with notations
	result := stringBuilder.Reset().
		AddAnyBit(
			anyBit := byteVar, 
			option := E_AddAnyBitOptions.BINARY, 
			lowerCase := FALSE, 
			displayedDigitsCount := 8, 
			addNotation := TRUE)
		.Create();
		
	AssertEquals_STRING(
		Actual := result,
		Expected := '(BIN)10101011',
		Message := 'Adding byte as BINARY with addNotation = TRUE was incorrect');
		
	// BINARY without notations
	result := stringBuilder.Reset()
		.AddAnyBit(
			anyBit := byteVar, 
			option := E_AddAnyBitOptions.BINARY, 
			lowerCase := FALSE, 
			displayedDigitsCount := 8, 
			addNotation := FALSE)
		.Create();
		
	AssertEquals_STRING(
		Actual := result,
		Expected := '10101011',
		Message := 'Adding byte as BINARY with addNotation = FALSE was incorrect');
		
	// DECIMAL with notations
	result := stringBuilder.Reset()
		.AddAnyBit(
			anyBit := byteVar, 
			option := E_AddAnyBitOptions.DECIMAL, 
			lowerCase := FALSE, 
			displayedDigitsCount := 8, 
			addNotation := TRUE)
		.Create();
		
	AssertEquals_STRING(
		Actual := result,
		Expected := '(DEC)00000171',
		Message := 'Adding byte as DECIMAL with addNotation = TRUE was incorrect');
		
	// DECIMAL without notations
	result := stringBuilder.Reset()
		.AddAnyBit(
			anyBit := byteVar, 
			option := E_AddAnyBitOptions.DECIMAL, 
			lowerCase := FALSE, 
			displayedDigitsCount := 8, 
			addNotation := FALSE)
		.Create();
		
	AssertEquals_STRING(
		Actual := result,
		Expected := '00000171',
		Message := 'Adding byte as DECIMAL with addNotation = FALSE was incorrect');

	// HEXADECIMAL with notations
	result := stringBuilder.Reset()
		.AddAnyBit(
			anyBit := byteVar, 
			option := E_AddAnyBitOptions.HEXADECIMAL, 
			lowerCase := FALSE, 
			displayedDigitsCount := 8, 
			addNotation := TRUE)
		.Create();
		
	AssertEquals_STRING(
		Actual := result,
		Expected := '(HEX)000000AB',
		Message := 'Adding byte as HEXADECIMAL with addNotation = TRUE was incorrect');
		
	// HEXADECIMAL without notations
	result := stringBuilder.Reset()
		.AddAnyBit(
			anyBit := byteVar, 
			option := E_AddAnyBitOptions.HEXADECIMAL, 
			lowerCase := FALSE, 
			displayedDigitsCount := 8, 
			addNotation := FALSE)
		.Create();
		
	AssertEquals_STRING(
		Actual := result,
		Expected := '000000AB',
		Message := 'Adding byte as HEXADECIMAL with addNotation = FALSE was incorrect');
	
	// OCTAL with notations
	result := stringBuilder.Reset()
		.AddAnyBit(
			anyBit := byteVar, 
			option := E_AddAnyBitOptions.OCTAL, 
			lowerCase := FALSE, 
			displayedDigitsCount := 8, 
			addNotation := TRUE)
		.Create();
		
	AssertEquals_STRING(
		Actual := result,
		Expected := '(OCT)00000253',
		Message := 'Adding byte as OCTAL with addNotation = TRUE was incorrect');
		
	// OCTAL without notations
	result := stringBuilder.Reset()
		.AddAnyBit(
			anyBit := byteVar, 
			option := E_AddAnyBitOptions.OCTAL, 
			lowerCase := FALSE, 
			displayedDigitsCount := 8, 
			addNotation := FALSE)
		.Create();
		
	AssertEquals_STRING(
		Actual := result,
		Expected := '00000253',
		Message := 'Adding byte as OCTAL with addNotation = FALSE was incorrect');
		
	TcUnit.TEST_FINISHED();
END_IF
END_METHOD

METHOD Test26_ANY_BIT_DWORD
VAR
	dwordVar	: DWORD := 16#AB;
	result	: Tc2_System.T_MaxString;
END_VAR
IF TcUnit.TEST_ORDERED('Test26_ANY_BIT_DWORD') THEN
	
	// BINARY with notations
	result := stringBuilder.Reset().
		AddAnyBit(
			anyBit := dwordVar, 
			option := E_AddAnyBitOptions.BINARY, 
			lowerCase := FALSE, 
			displayedDigitsCount := 32, 
			addNotation := TRUE)
		.Create();
		
	AssertEquals_STRING(
		Actual := result,
		Expected := '(BIN)00000000000000000000000010101011',
		Message := 'Adding dword as BINARY with addNotation = TRUE was incorrect');
		
	// BINARY without notations
	result := stringBuilder.Reset()
		.AddAnyBit(
			anyBit := dwordVar, 
			option := E_AddAnyBitOptions.BINARY, 
			lowerCase := FALSE, 
			displayedDigitsCount := 32, 
			addNotation := FALSE)
		.Create();
		
	AssertEquals_STRING(
		Actual := result,
		Expected := '00000000000000000000000010101011',
		Message := 'Adding dword as BINARY with addNotation = FALSE was incorrect');
		
	// DECIMAL with notations
	result := stringBuilder.Reset()
		.AddAnyBit(
			anyBit := dwordVar, 
			option := E_AddAnyBitOptions.DECIMAL, 
			lowerCase := FALSE, 
			displayedDigitsCount := 32, 
			addNotation := TRUE)
		.Create();
		
	AssertEquals_STRING(
		Actual := result,
		Expected := '(DEC)00000000000000000000000000000171',
		Message := 'Adding dword as DECIMAL with addNotation = TRUE was incorrect');
		
	// DECIMAL without notations
	result := stringBuilder.Reset()
		.AddAnyBit(
			anyBit := dwordVar, 
			option := E_AddAnyBitOptions.DECIMAL, 
			lowerCase := FALSE, 
			displayedDigitsCount := 32, 
			addNotation := FALSE)
		.Create();
		
	AssertEquals_STRING(
		Actual := result,
		Expected := '00000000000000000000000000000171',
		Message := 'Adding dword as DECIMAL with addNotation = FALSE was incorrect');

	// HEXADECIMAL with notations
	result := stringBuilder.Reset()
		.AddAnyBit(
			anyBit := dwordVar, 
			option := E_AddAnyBitOptions.HEXADECIMAL, 
			lowerCase := FALSE, 
			displayedDigitsCount := 32, 
			addNotation := TRUE)
		.Create();
		
	AssertEquals_STRING(
		Actual := result,
		Expected := '(HEX)000000000000000000000000000000AB',
		Message := 'Adding dword as HEXADECIMAL with addNotation = TRUE was incorrect');
		
	// HEXADECIMAL without notations
	result := stringBuilder.Reset()
		.AddAnyBit(
			anyBit := dwordVar, 
			option := E_AddAnyBitOptions.HEXADECIMAL, 
			lowerCase := FALSE, 
			displayedDigitsCount := 32, 
			addNotation := FALSE)
		.Create();
		
	AssertEquals_STRING(
		Actual := result,
		Expected := '000000000000000000000000000000AB',
		Message := 'Adding dword as HEXADECIMAL with addNotation = FALSE was incorrect');
	
	// OCTAL with notations
	result := stringBuilder.Reset()
		.AddAnyBit(
			anyBit := dwordVar, 
			option := E_AddAnyBitOptions.OCTAL, 
			lowerCase := FALSE, 
			displayedDigitsCount := 32, 
			addNotation := TRUE)
		.Create();
		
	AssertEquals_STRING(
		Actual := result,
		Expected := '(OCT)00000000000000000000000000000253',
		Message := 'Adding dword as OCTAL with addNotation = TRUE was incorrect');
		
	// OCTAL without notations
	result := stringBuilder.Reset()
		.AddAnyBit(
			anyBit := dwordVar, 
			option := E_AddAnyBitOptions.OCTAL, 
			lowerCase := FALSE, 
			displayedDigitsCount := 32, 
			addNotation := FALSE)
		.Create();
		
	AssertEquals_STRING(
		Actual := result,
		Expected := '00000000000000000000000000000253',
		Message := 'Adding dword as OCTAL with addNotation = FALSE was incorrect');
		
	TcUnit.TEST_FINISHED();
END_IF
END_METHOD

METHOD Test27_ANY_BIT_LWORD
VAR
	lwordVar	: LWORD := 16#AB;
	result	: Tc2_System.T_MaxString;
END_VAR
IF TcUnit.TEST_ORDERED('Test27_ANY_BIT_LWORD') THEN
	
	// BINARY with notations
	result := stringBuilder.Reset().
		AddAnyBit(
			anyBit := lwordVar, 
			option := E_AddAnyBitOptions.BINARY, 
			lowerCase := FALSE, 
			displayedDigitsCount := 64, 
			addNotation := TRUE)
		.Create();
		
	AssertEquals_STRING(
		Actual := result,
		Expected := '(BIN)0000000000000000000000000000000000000000000000000000000010101011',
		Message := 'Adding lword as BINARY with addNotation = TRUE was incorrect');
		
	// BINARY without notations
	result := stringBuilder.Reset()
		.AddAnyBit(
			anyBit := lwordVar, 
			option := E_AddAnyBitOptions.BINARY, 
			lowerCase := FALSE, 
			displayedDigitsCount := 64, 
			addNotation := FALSE)
		.Create();
		
	AssertEquals_STRING(
		Actual := result,
		Expected := '0000000000000000000000000000000000000000000000000000000010101011',
		Message := 'Adding lword as BINARY with addNotation = FALSE was incorrect');
		
	// DECIMAL with notations
	result := stringBuilder.Reset()
		.AddAnyBit(
			anyBit := lwordVar, 
			option := E_AddAnyBitOptions.DECIMAL, 
			lowerCase := FALSE, 
			displayedDigitsCount := 64, 
			addNotation := TRUE)
		.Create();
		
	AssertEquals_STRING(
		Actual := result,
		Expected := '(DEC)0000000000000000000000000000000000000000000000000000000000000171',
		Message := 'Adding lword as DECIMAL with addNotation = TRUE was incorrect');
		
	// DECIMAL without notations
	result := stringBuilder.Reset()
		.AddAnyBit(
			anyBit := lwordVar, 
			option := E_AddAnyBitOptions.DECIMAL, 
			lowerCase := FALSE, 
			displayedDigitsCount := 64, 
			addNotation := FALSE)
		.Create();
		
	AssertEquals_STRING(
		Actual := result,
		Expected := '0000000000000000000000000000000000000000000000000000000000000171',
		Message := 'Adding lword as DECIMAL with addNotation = FALSE was incorrect');

	// HEXADECIMAL with notations
	result := stringBuilder.Reset()
		.AddAnyBit(
			anyBit := lwordVar, 
			option := E_AddAnyBitOptions.HEXADECIMAL, 
			lowerCase := FALSE, 
			displayedDigitsCount := 64, 
			addNotation := TRUE)
		.Create();
		
	AssertEquals_STRING(
		Actual := result,
		Expected := '(HEX)00000000000000000000000000000000000000000000000000000000000000AB',
		Message := 'Adding lword as HEXADECIMAL with addNotation = TRUE was incorrect');
		
	// HEXADECIMAL without notations
	result := stringBuilder.Reset()
		.AddAnyBit(
			anyBit := lwordVar, 
			option := E_AddAnyBitOptions.HEXADECIMAL, 
			lowerCase := FALSE, 
			displayedDigitsCount := 64, 
			addNotation := FALSE)
		.Create();
		
	AssertEquals_STRING(
		Actual := result,
		Expected := '00000000000000000000000000000000000000000000000000000000000000AB',
		Message := 'Adding lword as HEXADECIMAL with addNotation = FALSE was incorrect');
	
	// OCTAL with notations
	result := stringBuilder.Reset()
		.AddAnyBit(
			anyBit := lwordVar, 
			option := E_AddAnyBitOptions.OCTAL, 
			lowerCase := FALSE, 
			displayedDigitsCount := 64, 
			addNotation := TRUE)
		.Create();
		
	AssertEquals_STRING(
		Actual := result,
		Expected := '(OCT)0000000000000000000000000000000000000000000000000000000000000253',
		Message := 'Adding lword as OCTAL with addNotation = TRUE was incorrect');
		
